PROGRAM UserMode
VAR
(*GapMode*)
	UserGapPositionNew:LREAL:=20;//target
	UserGapVelocityNew:LREAL:=0.02;//target
	UserGapPositionDisplay:LREAL;//current
	UserGapVelocityDisplay:LREAL;//current
(*ID taper mode*)
	UserTaperPositionNew:LREAL:=0;//target
	UserTaperVelocityNew:LREAL:=0.02;//target
	UserTaperPositionDisplay:LREAL;//current
	UserTaperPositionDisplayBLSide:LREAL;//current BeamLine
	UserTaperPositionActual:LREAL;//current
	UserTaperVelocityDisplay:LREAL;//target
	UserGapPositionDisplay_FromLeftTop:LREAL;
	UserGapPositionDisplay_FromLeftBottom:LREAL;
		//
	UserRightGapPositionNew:LREAL;
	UserRightGapVelocityNew:LREAL;
	UserRightGapPositionDisplay:LREAL;
	UserRightGapVelocityDisplay:LREAL;
	UserRightGapPositionDisplay_FromRightTop:LREAL;
	UserRightGapPositionDisplay_FromRightBottom:LREAL;
(*BL taper mode*)
	BLUserTaperPositionNew:LREAL:=0;//target
	BLUserTaperVelocityNew:LREAL:=0.02;//target
	BLUserTaperPositionDisplay:LREAL;//current
	//BLUserTaperPositionDisplayBLSide:LREAL;//current BeamLine
	BLUserTaperPositionActual:LREAL;//current
	BLUserTaperVelocityDisplay:LREAL;//target
	BLUserGapPositionDisplay_FromLeftTop:LREAL;
	BLUserGapPositionDisplay_FromLeftBottom:LREAL;
	//
	BLUserLeftGapPositionNew:LREAL;
	BLUserLeftGapVelocityNew:LREAL;
	BLUserLeftGapPositionDisplay:LREAL;
	BLUserLeftGapVelocityDisplay:LREAL;
	BLUserLeftGapPositionDisplay_FromLeftTop:LREAL;
	BLUserLeftGapPositionDisplay_FromLeftBottom:LREAL;
	BLUserRightGapPositionNew:LREAL;
	BLUserRightGapVelocityNew:LREAL;
	BLUserRightGapPositionDisplay:LREAL;
	BLUserRightGapVelocityDisplay:LREAL;
	BLUserRightGapPositionDisplay_FromRightTop:LREAL;
	BLUserRightGapPositionDisplay_FromRightBottom:LREAL;

	(**)
	btn_UserGapMove:BOOL;
	btn_UserGapStop:BOOL;
	(*Var*)
	fb_ton1:TON;
	fb_ton2:TON;
	fb_ton3:TON;
	(*Status*)
	State:DINT;
	Busy:BOOL;
	InitPowerDone:BOOL;
	InitCompensationDatasDone:BOOL;
	(*FB*)
	m_state: DINT;
	n_state: DINT;
	s_state: DINT;
	(*¼ì²âµ½ÏÞÎ»£¬»Ö¸´Move×´Ì¬*)
	FTrig_ReachLS: F_TRIG;
	FTrig_btn_GapMove: F_TRIG;
	GapOutRange: BOOL;
	(*PowerOff*)
	d_state: DINT;
	i: INT;
	j: INT;
	k: INT;
	moni_State:DINT;
	TargetPosLessThanCurrentPos:BOOL;
	TargetLTPosLessThanCurrentLTPos:BOOL;
	TargetRTPosLessThanCurrentRTPos:BOOL;
	TargetLBPosLessThanCurrentLBPos:BOOL;
	TargetRBPosLessThanCurrentRBPos:BOOL;
	PositiveMoving:BOOL;
	HysteresisMoving:BOOL;
	NoneHysteresisMoving:BOOL;
	(*Spectroscopy scanning Mode*)
	IsSSMotionMode:BOOL;
	RegularMotionMode:BOOL;
	SSMotionMode:BOOL;
	SS_StepSize:LREAL:=0.001;
	SS_StepNumber:INT:=10;
	SS_StepVelocity:LREAL:=1;
	SS_Move:BOOL;
	SS_Stop:BOOL;
	SS_MoveState:DINT;
	SS_StopState:DINT;
	SS_currentStep:DINT:=0;
	SS_StepSystemTime_Begin:ARRAY[0..100] OF ULINT;
	SS_StepSystemTime_End:ARRAY[0..100] OF ULINT;
	SS_StepCountTime:ARRAY[0..100] OF ULINT;
	SS_TimeCountBegin:BOOL;
	m: INT;
	SS_TON: TON;
	StepEachTime:TIME;
	StepEachTime_ms:INT:=1000;//ms
	SS_OTSTRUCT :OTSTRUCT ;
	SS_StartPositionDisplay:LREAL;
	RTRG_SS_StartPositionDisplay:R_TRIG;
	SS_InitStartPositionDone:BOOL;

	//
	min_SS_StepSize	: LREAL:=0;
	max_SS_StepSize	: LREAL:=200;
	inRange_SS_StepSize	: BOOL;
	//
	min_SS_StepNumber	: INT:=1;
	max_SS_StepNumber	: INT:=1000;
	inRange_SS_StepNumber	: BOOL;
	//
	min_SS_StepVelocity:LREAL:=0;
	max_SS_StepVelocity:LREAL:=1;
	inRange_SS_StepVelocity:BOOL;
	//
	min_StepEachTime_ms:INT:=100;
	max_StepEachTime_ms:INT:=10000;
	inRange_StepEachTime_ms:BOOL;
	l: INT;
	Threshold_UserTopPos_PLC: LREAL;
	Threshold_UserTopVelo_PLC: LREAL;
	Threshold_UserBottomPos_PLC: LREAL;
	Threshold_UserBottomVelo_PLC: LREAL;
	Threshold_UserLeftPos_PLC: LREAL;
	Threshold_UserLeftVelo_PLC: LREAL;
	Threshold_UserRightPos_PLC: LREAL;
	Threshold_UserRightVelo_PLC: LREAL;
	testa: BOOL;
	testb: BOOL;
	//Taper parameters
	Threshold_GapChangeFlag: LREAL:=0.001;
	Threshold_TaperChangeFlag: LREAL:=0.005;
	TaperAndGapSafetyfactor: LREAL:=1;
	TaperAndGapSafetyScale:LREAL:=0.41;//IAU=0.409,IVU=0.32,CPMU=0.328,IAMW=0.42
	TaperAndGapSafetyMinGapMargin:LREAL:=0.2;
	IDTaperAndBLTaperScale:LREAL:=0.548;//HU 
	//HEPSIDTaperAndBLTaperScale:LREAL:=0.55;
	//
	//Global Chain protection-MPS
	Global_ChainProtection_MPS_StorageRingReady:BOOL;
	Global_ChainProtection_MPS_On: BOOL;
	Global_ChainProtection_MPS_MaxGapValue: LREAL;
	Global_ChainProtection_MPS_MoveVelocity: LREAL;
	Global_ChainProtection_MPS_Done: BOOL;
	//Global_ChainProtection_Error: BOOL;
	//Global_ChainProtection_ErrorID: INT;
	//Global_ChainProtection_ErrorDescription: STRING;
	Global_ChainProtection_MPS_ManualOperation:BOOL:=TRUE;
	Global_ChainProtection_MPS_FTRIG:F_TRIG;
	Global_ChainProtection_MPS_FTRIG_Manul:F_TRIG;
	Global_ChainProtection_MPS_TON:TON;
	Global_ChainProtection_MPS_Triggered:BOOL;
	Global_ChainProtection_MPS_In:BOOL;
	Global_ChainProtection_MPS_In1 AT%I* :BOOL;//下降沿表示触发,EL1008
	Global_ChainProtection_MPS_In2 AT%I* :BOOL;
	Global_ChainProtection_MPS_State:DINT;
	Global_ChainProtection_MPS_Out1 AT%Q* :BOOL;//上升沿标识到达最大间隙，连锁保护成功,EL2624
	Global_ChainProtection_MPS_Out2 AT%Q* :BOOL;
	Global_ChainProtection_MPS_TON_Stop2Move:TON;
	Global_ChainProtection_MPS_TON_Stop2Move_InTaperMode:TON;
	Global_ChainProtection_MPS_TON_Power2Move:TON;
	//Global Chain protection-EPS
	Global_ChainProtection_EPS_BeamLineReady:BOOL;
	Global_ChainProtection_EPS_On: BOOL;
	Global_ChainProtection_EPS_MaxGapValue: LREAL;
	Global_ChainProtection_EPS_MoveVelocity: LREAL;
	Global_ChainProtection_EPS_Done: BOOL;
	//Global_ChainProtection_Error: BOOL;
	//Global_ChainProtection_ErrorID: INT;
	//Global_ChainProtection_ErrorDescription: STRING;
	Global_ChainProtection_EPS_ManualOperation:BOOL:=TRUE;
	Global_ChainProtection_EPS_FTRIG:F_TRIG;
	Global_ChainProtection_EPS_FTRIG_Manul:F_TRIG;
	Global_ChainProtection_EPS_TON:TON;
	Global_ChainProtection_EPS_Triggered:BOOL;
	Global_ChainProtection_EPS_In:BOOL;
	Global_ChainProtection_EPS_In1 AT%I* :BOOL;//下降沿表示触发,EL1124
	Global_ChainProtection_EPS_In2 AT%I* :BOOL;
	Global_ChainProtection_EPS_State:DINT;
	Global_ChainProtection_EPS_Out1 AT%Q* :BOOL;//上升沿标识到达最大间隙，连锁保护成功,EL2124
	Global_ChainProtection_EPS_Out2 AT%Q* :BOOL;
	Global_ChainProtection_EPS_TON_Stop2Move:TON;
	Global_ChainProtection_EPS_TON_Stop2Move_InTaperMode:TON;
	Global_ChainProtection_EPS_TON_Power2Move:TON;
	//
	//Cryogenic Chain protection
	Cryogenic_ChainProtection_On: BOOL;
	Cryogenic_ChainProtection_MaxGapValue: LREAL;
	Cryogenic_ChainProtection_MoveVelocity: LREAL;
	Cryogenic_ChainProtection_Done: BOOL;
	//Cryogenic_ChainProtection_Error: BOOL;
	//Cryogenic_ChainProtection_ErrorID: INT;
	//Cryogenic_ChainProtection_ErrorDescription: STRING;
	Cryogenic_ChainProtection_ManualOperation:BOOL:=TRUE;
	Cryogenic_ChainProtection_FTRIG:F_TRIG;
	Cryogenic_ChainProtection_FTRIG_Manul:F_TRIG;
	Cryogenic_ChainProtection_TON:TON;
	Cryogenic_ChainProtection_Triggered:BOOL;
	Cryogenic_ChainProtection_In:BOOL;
	Cryogenic_ChainProtection_State:DINT;
	Cryogenic_ChainProtection_Out1 AT%Q* :BOOL;//上升沿标识到达最大间隙，连锁保护成功
	Cryogenic_ChainProtection_TON_Stop2Move:TON;
	Cryogenic_ChainProtection_TON_Stop2Move_InTaperMode:TON;
	Cryogenic_ChainProtection_TON_Power2Move:TON;
	test11:INT:=1;
	IsTest11OrNot:BOOL;
	tesetBegin: BOOL;
	Threshold_motorsTargetPosCalculate: LREAL;
	SS_Stop2: BOOL;
	//
	LeftTopLinPositionNewTemp: LREAL;
	RightTopLinPositionNewTemp: LREAL;
	LeftBottomLinPositionNewTemp: LREAL;
	RightBottomLinPositionNewTemp: LREAL;
	
	
	//OneKeyToMaxGap
	btn_OneKeyToMaxGap:BOOL;
	OneKeyToMaxGap_RTRIG:R_TRIG;
	OneKeyToMaxGap_TON:TON;
	OneKeyToMaxGap_Triggered:BOOL;
	OneKeyToMaxGap_State:DINT;
	OneKeyToMaxGap_TON_Stop2Move:TON;
	OneKeyToMaxGap_TON_Stop2Move_InTaperMode:TON;
	OneKeyToMaxGap_TON_Power2Move:TON;
	OneKeyToMaxGap_Done:BOOL;
	FTrig_ReachLSa: F_TRIG;
	Unreach_LS_Fara: BOOL;
	Unreach_LS_Neara: BOOL;
	btn_UserGapStopa: BOOL;
	
	//OneKeyToMTaperZero
	btn_OneKeyToTaperZero:BOOL;
	OneKeyToTaperZero_RTRIG:R_TRIG;
	OneKeyToTaperZero_TON:TON;
	OneKeyToTaperZero_Triggered:BOOL;
	OneKeyToTaperZero_State:DINT;
	OneKeyToTaperZero_Done:BOOL;
	OneKeyToTaperZero_Delay:TON;
	//BLTaper
	CurrentTaperInit: LREAL;
	L_HalfGirder:LREAL:=2500;
	L_Center2Motor:LREAL:=1375;
	
	trig_TaperOrNot: R_TRIG;
	trig_BLTaperOrNot: R_TRIG;
END_VAR

IF NOT PositionBiasDone THEN
	RETURN;
END_IF
IF NOT loadParametersDone THEN
	RETURN;
END_IF
(*btn_Power On/Off*)
IF btn_Power AND NOT st_Power THEN
	btn_PowerOn:=TRUE;
	btn_Power:=FALSE;
END_IF
IF btn_Power AND st_Power THEN
	btn_PowerOff:=TRUE;
	btn_Power:=FALSE;
END_IF
IF btn_PowerOn THEN
	A_PowerOn();
END_IF
IF btn_PowerOff THEN
	A_PowerOff();
END_IF

(*检查couple状态，不允许couple*)
A_CheckCoupleStatus();

(*监控四轴位置速度等*)
A_MonitoringAllAxis();

(*目标位置和速度保护*)
A_CheckMotorsPos();

(*补偿数据处理*)
A_InitCompensationData();

(*常规磁间隙开合*)
IF RegularMotionMode AND NOT SSMotionMode THEN
	A_RegularMotion();
END_IF

(*Spectroscopy scanning Mode*)
IF IsSSMotionMode THEN
	SSMotionMode:=TRUE;
	RegularMotionMode:=FALSE;
ELSE
	SSMotionMode:=FALSE;
	RegularMotionMode:=TRUE;
END_IF
IF	SSMotionMode AND NOT RegularMotionMode THEN
	A_SpectroscopyScanningMotion();
END_IF


(*GlobalChainProtection*)
A_GlobalChainProtection_MPS();
A_GlobalChainProtection_EPS();

(*CryogenicChainProtection*)
A_CryogenicChainProtection();

(*A_OneKeyToMaxGap*)
A_OneKeyToMaxGap();

(*A_OneKeyToTaperZero*)
A_OneKeyToTaperZero();

(*A_TaperParametersInit*)
A_TaperParametersInit();

ACTION A_CheckCoupleStatus:
IF NOT btn_PowerOff THEN
	IF st_Power=1 AND st_Couple<>0THEN
		Error:=TRUE;
		ErrorID:=501;
		LeftTopLinMoveIndicator:=0;
		RightTopLinMoveIndicator:=0;
		LeftBottomLinMoveIndicator:=0;
		RightBottomLinMoveIndicator:=0;
		FB_PlcEmergencyStop();
		LED_Error:=TRUE;
		ErrorDescription:='couple stutas error';
	END_IF
END_IF
END_ACTION

ACTION A_CheckMotorsPos:
//
//目标位置速度超出阈值判断
//
//gap posiion
IF UserGapPositionNew<min_UserGapPositionNew OR UserGapPositionNew>max_UserGapPositionNew THEN
	inRange_UserGapPositionNew:=FALSE;
END_IF
IF UserGapPositionNew>=min_UserGapPositionNew AND UserGapPositionNew<=max_UserGapPositionNew THEN
	inRange_UserGapPositionNew:=TRUE;
END_IF
//gap velocity
IF UserGapVelocityNew<min_UserGapVelocityNew OR UserGapVelocityNew>max_UserGapVelocityNew THEN
	inRange_UserGapVelocityNew:=FALSE;
END_IF
IF UserGapVelocityNew>=min_UserGapVelocityNew AND UserGapVelocityNew<=max_UserGapVelocityNew THEN
	inRange_UserGapVelocityNew:=TRUE;
END_IF
//taper position
IF UserTaperPositionNew<min_UserTaperPositionNew OR UserTaperPositionNew>max_UserTaperPositionNew THEN
	inRange_UserTaperPositionNew:=FALSE;
END_IF
IF UserTaperPositionNew>=min_UserTaperPositionNew AND UserTaperPositionNew<=max_UserTaperPositionNew THEN
	inRange_UserTaperPositionNew:=TRUE;
END_IF
//taper velocity
IF UserTaperVelocityNew<min_UserTaperVelocityNew OR UserTaperVelocityNew>max_UserTaperVelocityNew THEN
	inRange_UserTaperVelocityNew:=FALSE;
END_IF
IF UserTaperVelocityNew>=min_UserTaperVelocityNew AND UserTaperVelocityNew<=max_UserTaperVelocityNew THEN
	inRange_UserTaperVelocityNew:=TRUE;
END_IF
//SS Mode
IF SS_StepSize<min_SS_StepSize OR SS_StepSize>max_SS_StepSize THEN
	inRange_SS_StepSize:=FALSE;
END_IF
IF SS_StepSize>=min_SS_StepSize AND SS_StepSize<=max_SS_StepSize THEN
	inRange_SS_StepSize:=TRUE;
END_IF
IF SS_StepNumber<min_SS_StepNumber OR SS_StepNumber>max_SS_StepNumber THEN
	inRange_SS_StepNumber:=FALSE;
END_IF
IF SS_StepNumber>=min_SS_StepNumber AND SS_StepNumber<=max_SS_StepNumber THEN
	inRange_SS_StepNumber:=TRUE;
END_IF
IF SS_StepVelocity<min_SS_StepVelocity OR SS_StepVelocity>max_SS_StepVelocity THEN
	inRange_SS_StepVelocity:=FALSE;
END_IF
IF SS_StepVelocity>=min_SS_StepVelocity AND SS_StepVelocity<=max_SS_StepVelocity THEN
	inRange_SS_StepVelocity:=TRUE;
END_IF
IF StepEachTime_ms<min_StepEachTime_ms OR StepEachTime_ms>max_StepEachTime_ms THEN
	inRange_StepEachTime_ms:=FALSE;
END_IF
IF StepEachTime_ms>=min_StepEachTime_ms AND StepEachTime_ms<=max_StepEachTime_ms THEN
	inRange_StepEachTime_ms:=TRUE;
END_IF


//
//输入速度和位置保护
//
IF btn_UserGapMove  AND NOT SSMotionMode AND RegularMotionMode THEN
	IF NOT inRange_UserGapPositionNew THEN
		btn_UserGapStop:=TRUE;
		btn_UserGapMove:=FALSE;
		Error:=TRUE;
		ErrorId:=801;
		ErrorDescription:='target Gap position out of range,please check';
		RETURN;
	ELSE
		//btn_UserGapStop:=FALSE;
		Error:=FALSE;
		ErrorId:=0;
		ErrorDescription:='';	
	END_IF
	IF NOT inRange_UserGapVelocityNew THEN
		btn_UserGapStop:=TRUE;
		btn_UserGapMove:=FALSE;
		Error:=TRUE;
		ErrorId:=802;
		ErrorDescription:='target Gap velocity out of range,please check';
		RETURN;
	ELSE
		//btn_UserGapStop:=FALSE;
		Error:=FALSE;
		ErrorId:=0;
		ErrorDescription:='';
	END_IF
	IF NOT inRange_UserTaperPositionNew THEN
		btn_UserGapStop:=TRUE;
		btn_UserGapMove:=FALSE;
		Error:=TRUE;
		ErrorId:=803;
		ErrorDescription:='target Taper Position out of range,please check';
		RETURN;
	ELSE
		//btn_UserGapStop:=FALSE;
		Error:=FALSE;
		ErrorId:=0;
		ErrorDescription:='';
	END_IF
	IF NOT inRange_UserTaperVelocityNew THEN
		btn_UserGapStop:=TRUE;
		btn_UserGapMove:=FALSE;
		Error:=TRUE;
		ErrorId:=804;
		ErrorDescription:='target Taper velocity out of range,please check';
		RETURN;
	ELSE
		//btn_UserGapStop:=FALSE;
		Error:=FALSE;
		ErrorId:=0;
		ErrorDescription:='';
	END_IF
END_IF

//
//运动过程中，监控目标位置速度
//
IF moveStatusAnyAxis THEN
	IF NOT inRange_UserGapPositionNew THEN
		btn_UserGapStop:=TRUE;
		Error:=TRUE;
		ErrorId:=805;
		ErrorDescription:='target Gap position out of range in moving process!';
		FB_PlcEmergencyStop();
	END_IF
	IF NOT inRange_UserGapVelocityNew THEN
		btn_UserGapStop:=TRUE;
		Error:=TRUE;
		ErrorId:=806;
		ErrorDescription:='target Gap velocity out of range in moving process!';
		FB_PlcEmergencyStop();
	END_IF
	IF NOT inRange_UserTaperPositionNew THEN
		btn_UserGapStop:=TRUE;
		Error:=TRUE;
		ErrorId:=807;
		ErrorDescription:='target Taper Position out of range in moving process!';
		FB_PlcEmergencyStop();
	END_IF
	IF NOT inRange_UserTaperVelocityNew THEN
		btn_UserGapStop:=TRUE;
		Error:=TRUE;
		ErrorId:=808;
		ErrorDescription:='target Taper velocity out of range in moving process!';
		FB_PlcEmergencyStop();
	END_IF
END_IF
//
//运动过程中，监控每一个轴的目标位置，目标位置若超出阈值，Emergency
//
IF moveStatusAnyAxis THEN
	IF NOT TaperOrNot THEN
		IF LeftTopLinPositionNew<min_UserLEProtectionGapPosition/2 OR LeftTopLinPositionNew>max_UserLEProtectionGapPosition/2 THEN
			btn_UserGapStop:=TRUE;
			Error:=TRUE;
			ErrorId:=809;
			ErrorDescription:='target LeftTop position out of range in moving process!';
			FB_PlcEmergencyStop();
		END_IF
		IF RightTopLinPositionNew<min_UserLEProtectionGapPosition/2 OR RightTopLinPositionNew>max_UserLEProtectionGapPosition/2 THEN
			btn_UserGapStop:=TRUE;
			Error:=TRUE;
			ErrorId:=810;
			ErrorDescription:='target RightTop velocity out of range in moving process!';
			FB_PlcEmergencyStop();
		END_IF
		IF LeftBottomLinPositionNew<min_UserLEProtectionGapPosition/2 OR LeftBottomLinPositionNew>max_UserLEProtectionGapPosition/2 THEN
			btn_UserGapStop:=TRUE;
			Error:=TRUE;
			ErrorId:=812;
			ErrorDescription:='target LeftBottom Position out of range in moving process!';
			FB_PlcEmergencyStop();
		END_IF
		IF RightBottomLinPositionNew<min_UserLEProtectionGapPosition/2 OR RightBottomLinPositionNew>max_UserLEProtectionGapPosition/2 THEN
			btn_UserGapStop:=TRUE;
			Error:=TRUE;
			ErrorId:=813;
			ErrorDescription:='target RightBottom Position out of range in moving process!';
			FB_PlcEmergencyStop();
		END_IF
	ELSE//Taper状态的保护
		;//Taper状态下，不用监控四轴位置，只需要监控目标Taper位置。在上面已经保护
	END_IF
END_IF
END_ACTION

ACTION A_CryogenicChainProtection:
//总开关
IF NOT Cryogenic_ChainProtection_On THEN
	RETURN;
END_IF
IF NOT MAIN.CryogenicCompensationOn THEN
	RETURN;
END_IF
//判断插入件状态，是否就位
//IF NOT IDControlReady THEN
//	Cryogenic_ChainProtection_Done:=FALSE;
//	Error:= TRUE;
//	ErrorID:=1501;
//	ErrorDescription:='ID NOT READY!';
//	RETURN;
//END_IF

//
//全局连锁保护程序开始
//
//0.检测温度变化超出正常范围，或者手动触发，触发低温联锁保护
//1.判断电机是否在开启状态,没有就打开电源
//2.判断是否在Moving状态,若有就Stop
//3.将磁间隙打开到至最大阈值
//4.到位后给出反馈，且安全PLC触发
//IF MAIN.temperatureStatus=3 THEN //=2低温,超出低温阈值就触发保护
//	Cryogenic_ChainProtection_Triggered:=TRUE;
//END_IF
Cryogenic_ChainProtection_FTRIG(CLK:=MAIN.InCryogenicOrNot);
IF Cryogenic_ChainProtection_FTRIG.Q THEN
	Cryogenic_ChainProtection_Triggered:=TRUE;
END_IF
Cryogenic_ChainProtection_FTRIG_Manul(CLK:=Cryogenic_ChainProtection_ManualOperation);
IF Cryogenic_ChainProtection_FTRIG_Manul.Q THEN
	Cryogenic_ChainProtection_Triggered:=TRUE;
END_IF
IF Cryogenic_ChainProtection_Triggered THEN
	//判断当前间隙，如果比Cryogenic_ChainProtection_MaxGapValue大，则不动作，只报警，且安全PLC触发
	IF UserGapPositionDisplay - Cryogenic_ChainProtection_MaxGapValue >=0.001THEN
		Cryogenic_ChainProtection_Done:=TRUE;
		Plc_EmergencyStop:=FALSE;
		Error:= TRUE;
		ErrorID:= 1502;
		ErrorDescription:='Cryogenic Abnormal !';
		RETURN;
	END_IF
	CASE Cryogenic_ChainProtection_State OF
		0://1.判断电机是否在开启状态,没有就打开电源
			IF st_Power=1 THEN
				Cryogenic_ChainProtection_State:=1;
			ELSE
				btn_PowerOn:=TRUE;
				IF btn_PowerOn THEN
					A_PowerOn();
				END_IF
			END_IF
		1://1.判断是否在谱学扫描模式，如果是，则切换回正常运动模式
			IF IsSSMotionMode THEN
				SS_Stop:=TRUE;
				IsSSMotionMode:=FALSE;
			END_IF
			Cryogenic_ChainProtection_State:=2;
		2://判断是否在taper，如果在taper,则判断是否在运动，如果是，则停止运动,0.5sh后，转入下一步
			IF TaperOrNot THEN
				IF moveStatusLeftTop OR moveStatusRightTop OR moveStatusLeftBottom OR moveStatusRightBottom THEN
					btn_UserGapStop:=TRUE;
				ELSE
					Cryogenic_ChainProtection_TON_Stop2Move_InTaperMode(PT:=T#0.5S);
					Cryogenic_ChainProtection_TON_Stop2Move_InTaperMode.IN:=TRUE;
					IF Cryogenic_ChainProtection_TON_Stop2Move_InTaperMode.Q THEN
						TaperOrNot:=FALSE;//关闭taper模式
						Cryogenic_ChainProtection_State:=3;
					END_IF
				END_IF
			ELSE
				Cryogenic_ChainProtection_State:=3;
			END_IF
		3://3.判断是否在Moving状态,若有就Stop.Taper模式已处理完，此处开始走正常GAP开合逻辑
			IF moveStatusLeftTop OR moveStatusRightTop OR moveStatusLeftBottom OR moveStatusRightBottom THEN
				btn_UserGapStop:=TRUE;
			ELSE
				Cryogenic_ChainProtection_TON_Stop2Move(PT:=T#0.5S);
				Cryogenic_ChainProtection_TON_Stop2Move.IN:=TRUE;
				IF Cryogenic_ChainProtection_TON_Stop2Move.Q THEN
					Cryogenic_ChainProtection_State:=4;
				END_IF
			END_IF
		4://4.将磁间隙打开到至最大阈值
			Cryogenic_ChainProtection_TON(PT:=INT_TO_TIME(LREAL_TO_INT(Cryogenic_ChainProtection_MaxGapValue/Cryogenic_ChainProtection_MoveVelocity+30))*1000);
			Cryogenic_ChainProtection_TON.IN:=TRUE;
			Cryogenic_ChainProtection_TON_Power2Move(PT:=T#0.1S);
			Cryogenic_ChainProtection_TON_Power2Move.IN:=TRUE;
			UserGapPositionNew:=Cryogenic_ChainProtection_MaxGapValue;
			UserGapVelocityNew:=Cryogenic_ChainProtection_MoveVelocity;
			btn_UserGapMove:=TRUE;
			IF Cryogenic_ChainProtection_TON_Power2Move.Q THEN
				IF FB_MOVE.BCGapDone THEN
					Cryogenic_ChainProtection_State:=88;
				END_IF
			END_IF
			IF Cryogenic_ChainProtection_TON.Q THEN//如果150s后，还没有运动到指定gap，则报错
				Cryogenic_ChainProtection_State:=-100;
			END_IF
		88://4.到位后给出反馈，且安全PLC触发
			Cryogenic_ChainProtection_Done:=TRUE;
			Plc_EmergencyStop:=FALSE;		
			Error:=TRUE;
			ErrorID:=1503;
			ErrorDescription:='Cryogenic_ChainProtection Triggered';
		-100:
			Cryogenic_ChainProtection_Done:=FALSE;
			Error:=TRUE;
			ErrorID:=1504;
			ErrorDescription:='NOT MOVING TO MAXGAP';
	END_CASE
END_IF

//监控是否同时是低温模式，且温度传感器检测到的是低温+10℃（避开低温联锁保护，联锁保护要求在低温阈值时拉开磁间隙）
IF MAIN.temperatureStatus<>0 AND MAIN.temperature_average > MAIN.CryogenicTemperatureThreshold +10 THEN//在低温+10℃
	IF MAIN.HasTemperatureSensorOrNot AND MAIN.CryogenicCompensationOn THEN
			Error:=TRUE;
			ErrorID:=1505;
			Plc_EmergencyStop:=FALSE;
			ErrorDescription:='CryogenicCompensationOn AND Room temperatureStatus';
	END_IF
END_IF
END_ACTION

ACTION A_GlobalChainProtection_EPS:
//硬线输入定义
Global_ChainProtection_EPS_In:=Global_ChainProtection_EPS_In1 AND Global_ChainProtection_EPS_In2;
//硬线输出定义
Global_ChainProtection_EPS_Out1:=Global_ChainProtection_EPS_Done;
Global_ChainProtection_EPS_Out2:=Global_ChainProtection_EPS_Done;
//总开关
IF NOT Global_ChainProtection_EPS_On THEN
	RETURN;
END_IF
//判断插入件状态，是否就位
//IF NOT IDControlReady THEN
//	Global_ChainProtection_EPS_Done:=FALSE;
//	Error:= TRUE;
//	ErrorID:= 1501;
//	ErrorDescription:='ID NOT READY!';
//	RETURN;
//END_IF
//判断储存环是否给出就位信号，暂时由参数表给出TRUE，最终将由IOC接受PV
IF 	NOT Global_ChainProtection_EPS_BeamLineReady THEN
	Global_ChainProtection_EPS_Done:=FALSE;
	Error:= TRUE;
	ErrorID:= 1503;
	ErrorDescription:='Global_ChainProtection_EPS_BeamLineReady NOT Ready';
	RETURN;
END_IF
//
//全局连锁保护程序开始
//
//0.检测到下降沿，触发
//1.判断电机是否在开启状态,没有就打开电源
//2.判断是否在Moving状态,若有就Stop
//3.将磁间隙打开到至最大阈值
//4.到位后给出反馈，且安全PLC触发
Global_ChainProtection_EPS_FTRIG(CLK:=Global_ChainProtection_EPS_In);
IF Global_ChainProtection_EPS_FTRIG.Q THEN
	Global_ChainProtection_EPS_Triggered:=TRUE;
END_IF
Global_ChainProtection_EPS_FTRIG_Manul(CLK:=Global_ChainProtection_EPS_ManualOperation);
IF Global_ChainProtection_EPS_FTRIG_Manul.Q THEN
	Global_ChainProtection_EPS_Triggered:=TRUE;
END_IF
IF Global_ChainProtection_EPS_Triggered THEN
	CASE Global_ChainProtection_EPS_State OF
		0://1.判断电机是否在开启状态,没有就打开电源
			IF st_Power=1 THEN
				Global_ChainProtection_EPS_State:=1;
			ELSE
				btn_PowerOn:=TRUE;
				IF btn_PowerOn THEN
					A_PowerOn();
				END_IF
			END_IF
		1://1.判断是否在谱学扫描模式，如果是，则切换回正常运动模式
			IF IsSSMotionMode THEN
				SS_Stop:=TRUE;
				IsSSMotionMode:=FALSE;
			END_IF
			Global_ChainProtection_EPS_State:=2;
		2://判断是否在taper，如果在taper,则判断是否在运动，如果是，则停止运动,0.5sh后，转入下一步
			IF TaperOrNot THEN
				IF moveStatusLeftTop OR moveStatusRightTop OR moveStatusLeftBottom OR moveStatusRightBottom THEN
					btn_UserGapStop:=TRUE;
				ELSE
					Global_ChainProtection_EPS_TON_Stop2Move_InTaperMode(PT:=T#0.5S);
					Global_ChainProtection_EPS_TON_Stop2Move_InTaperMode.IN:=TRUE;
					IF Global_ChainProtection_EPS_TON_Stop2Move_InTaperMode.Q THEN
						TaperOrNot:=FALSE;//关闭taper模式
						Global_ChainProtection_EPS_State:=3;
					END_IF
				END_IF
			ELSE
				Global_ChainProtection_EPS_State:=3;
			END_IF
		3://3.判断是否在Moving状态,若有就Stop.Taper模式已处理完，此处开始走正常GAP开合逻辑
			IF moveStatusLeftTop OR moveStatusRightTop OR moveStatusLeftBottom OR moveStatusRightBottom THEN
				btn_UserGapStop:=TRUE;
			ELSE
				Global_ChainProtection_EPS_TON_Stop2Move(PT:=T#0.5S);
				Global_ChainProtection_EPS_TON_Stop2Move.IN:=TRUE;
				IF Global_ChainProtection_EPS_TON_Stop2Move.Q THEN
					Global_ChainProtection_EPS_State:=4;
				END_IF
			END_IF
		4://当前磁间隙如何和最大磁间隙差别不大，不超过0.1，则直接保护
			IF ABS(UserGapPositionDisplay-Global_ChainProtection_EPS_MaxGapValue)<=0.1 THEN
				Global_ChainProtection_EPS_Done:=TRUE;
				Plc_EmergencyStop:=FALSE;	
				Error:=TRUE;
				ErrorID:=1506;
				ErrorDescription:='EPS Triggered,but ABS(GapPositionDisplay-EPS_MaxGapValue)<=0.1 ';	
			ELSE
				Global_ChainProtection_EPS_State:=5;
			END_IF
		5://5.将磁间隙打开到至最大阈值
			Global_ChainProtection_EPS_TON(PT:=INT_TO_TIME(LREAL_TO_INT(Global_ChainProtection_EPS_MaxGapValue/Global_ChainProtection_EPS_MoveVelocity+30))*1000);
			Global_ChainProtection_EPS_TON.IN:=TRUE;
			Global_ChainProtection_EPS_TON_Power2Move(PT:=T#0.1S);
			Global_ChainProtection_EPS_TON_Power2Move.IN:=TRUE;
			UserGapPositionNew:=Global_ChainProtection_EPS_MaxGapValue;
			UserGapVelocityNew:=Global_ChainProtection_EPS_MoveVelocity;
			btn_UserGapMove:=TRUE;
			IF Global_ChainProtection_EPS_TON_Power2Move.Q THEN
				IF FB_MOVE.BCGapDone THEN
					Global_ChainProtection_EPS_State:=88;
				END_IF
			END_IF
			IF Global_ChainProtection_EPS_TON.Q THEN//如果150s后，还没有运动到指定gap，则报错
				Global_ChainProtection_EPS_State:=-100;
			END_IF
		88://6.到位后给出反馈，且安全PLC触发
			Global_ChainProtection_EPS_Done:=TRUE;
			Plc_EmergencyStop:=FALSE;	
			Error:=TRUE;
			ErrorID:=1504;
			ErrorDescription:='Global_ChainProtection_EPS Triggered ';	
		-100:
			Global_ChainProtection_EPS_Done:=FALSE;
			Error:=TRUE;
			ErrorID:=1505;
			ErrorDescription:='NOT MOVING TO MAXGAP';
	END_CASE
END_IF
END_ACTION

ACTION A_GlobalChainProtection_MPS:
//硬线输入定义
Global_ChainProtection_MPS_In:=Global_ChainProtection_MPS_In1 AND Global_ChainProtection_MPS_In2;
//硬线输出定义
Global_ChainProtection_MPS_Out1:=Global_ChainProtection_MPS_Done;
Global_ChainProtection_MPS_Out2:=Global_ChainProtection_MPS_Done;
//总开关
IF NOT Global_ChainProtection_MPS_On THEN
	RETURN;
END_IF
//判断插入件状态，是否就位
//IF NOT IDControlReady THEN
//	Global_ChainProtection_MPS_Done:=FALSE;
//	Error:= TRUE;
//	ErrorID:= 1401;
//	ErrorDescription:='ID NOT READY!';
//	RETURN;
//END_IF
//判断储存环是否给出就位信号，暂时由参数表给出TRUE，最终将由IOC接受PV
IF 	NOT Global_ChainProtection_MPS_StorageRingReady THEN
	Global_ChainProtection_MPS_Done:=FALSE;
	Error:= TRUE;
	ErrorID:= 1403;
	ErrorDescription:='StorageRingChainProtection NOT Ready';
	RETURN;
END_IF
//
//全局连锁保护程序开始
//
//0.检测到下降沿，触发
//1.判断电机是否在开启状态,没有就打开电源
//2.判断是否在Moving状态,若有就Stop
//3.将磁间隙打开到至最大阈值
//4.到位后给出反馈，且安全PLC触发
Global_ChainProtection_MPS_FTRIG(CLK:=Global_ChainProtection_MPS_In);
IF Global_ChainProtection_MPS_FTRIG.Q THEN
	Global_ChainProtection_MPS_Triggered:=TRUE;
END_IF
Global_ChainProtection_MPS_FTRIG_Manul(CLK:=Global_ChainProtection_MPS_ManualOperation);
IF Global_ChainProtection_MPS_FTRIG_Manul.Q THEN
	Global_ChainProtection_MPS_Triggered:=TRUE;
END_IF
IF Global_ChainProtection_MPS_Triggered THEN
	CASE Global_ChainProtection_MPS_State OF
		0://1.判断电机是否在开启状态,没有就打开电源
			IF st_Power=1 THEN
				Global_ChainProtection_MPS_State:=1;
			ELSE
				btn_PowerOn:=TRUE;
				IF btn_PowerOn THEN
					A_PowerOn();
				END_IF
			END_IF
		1://1.判断是否在谱学扫描模式，如果是，则切换回正常运动模式
			IF IsSSMotionMode THEN
				SS_Stop:=TRUE;
				IsSSMotionMode:=FALSE;
			END_IF
			Global_ChainProtection_MPS_State:=2;
		2://判断是否在taper，如果在taper,则判断是否在运动，如果是，则停止运动,0.5sh后，转入下一步
			IF TaperOrNot THEN
				IF moveStatusLeftTop OR moveStatusRightTop OR moveStatusLeftBottom OR moveStatusRightBottom THEN
					btn_UserGapStop:=TRUE;
				ELSE
					Global_ChainProtection_MPS_TON_Stop2Move_InTaperMode(PT:=T#0.5S);
					Global_ChainProtection_MPS_TON_Stop2Move_InTaperMode.IN:=TRUE;
					IF Global_ChainProtection_MPS_TON_Stop2Move_InTaperMode.Q THEN
						TaperOrNot:=FALSE;//关闭taper模式
						Global_ChainProtection_MPS_State:=3;
					END_IF
				END_IF
			ELSE
				Global_ChainProtection_MPS_State:=3;
			END_IF
		3://3.判断是否在Moving状态,若有就Stop.Taper模式已处理完，此处开始走正常GAP开合逻辑
			IF moveStatusLeftTop OR moveStatusRightTop OR moveStatusLeftBottom OR moveStatusRightBottom THEN
				btn_UserGapStop:=TRUE;
			ELSE
				Global_ChainProtection_MPS_TON_Stop2Move(PT:=T#0.5S);
				Global_ChainProtection_MPS_TON_Stop2Move.IN:=TRUE;
				IF Global_ChainProtection_MPS_TON_Stop2Move.Q THEN
					Global_ChainProtection_MPS_State:=4;
				END_IF
			END_IF
		4://当前磁间隙如何和最大磁间隙差别不大，不超过0.1，则直接保护
			IF ABS(UserGapPositionDisplay-Global_ChainProtection_MPS_MaxGapValue)<=0.1 THEN
				Global_ChainProtection_MPS_Done:=TRUE;
				Plc_EmergencyStop:=FALSE;	
				Error:=TRUE;
				ErrorID:=1406;
				ErrorDescription:='MPS Triggered,but ABS(GapPositionDisplay-MPS_MaxGapValue)<=0.1 ';	
			ELSE
				Global_ChainProtection_MPS_State:=5;
			END_IF
		5://5.将磁间隙打开到至最大阈值
			Global_ChainProtection_MPS_TON(PT:=INT_TO_TIME(LREAL_TO_INT(Global_ChainProtection_MPS_MaxGapValue/Global_ChainProtection_MPS_MoveVelocity+30))*1000);
			Global_ChainProtection_MPS_TON.IN:=TRUE;
			Global_ChainProtection_MPS_TON_Power2Move(PT:=T#0.1S);
			Global_ChainProtection_MPS_TON_Power2Move.IN:=TRUE;
			UserGapPositionNew:=Global_ChainProtection_MPS_MaxGapValue;
			UserGapVelocityNew:=Global_ChainProtection_MPS_MoveVelocity;
			btn_UserGapMove:=TRUE;
			IF Global_ChainProtection_MPS_TON_Power2Move.Q THEN
				IF FB_MOVE.BCGapDone THEN
					Global_ChainProtection_MPS_State:=88;
				END_IF
			END_IF
			IF Global_ChainProtection_MPS_TON.Q THEN//如果150s后，还没有运动到指定gap，则报错
				Global_ChainProtection_MPS_State:=-100;
			END_IF
		88://6.到位后给出反馈，且安全PLC触发
			Global_ChainProtection_MPS_Done:=TRUE;
			Plc_EmergencyStop:=FALSE;	
			Error:=TRUE;
			ErrorID:=1404;
			ErrorDescription:='Global_ChainProtection_MPS Triggered ';	
		-100:
			Global_ChainProtection_MPS_Done:=FALSE;
			Error:=TRUE;
			ErrorID:=1405;
			ErrorDescription:='NOT MOVING TO MAXGAP';
	END_CASE
END_IF
END_ACTION

ACTION A_InitCompensationData:
(*补偿开始*)
IF USE_SingleAxis_Compensation THEN
(*正常gap模式以及插入件taper模式下，只运动出口电机，因此只解算出口位置*)
	IF NormalGapMode OR IDTaperMode THEN
		//
		//1.目标位置解算
		//
		(*通过补偿表解算四轴目标位置*)
		//左轴位置由Gap定，右轴位置由右gap定。右gap值=左gap+taper。taper模式和非taper模式一样，非taper模式只是一种特例存在
		//左轴目标位置解算
		IF NOT TaperOrNot THEN
			UserTaperPositionNew:=0;
			//UserTaperPositionDisplay:=0;
		END_IF
		UserRightGapPositionNew:=UserGapPositionNew+UserTaperPositionNew;
		//左轴目标位置解算
		FOR	i:= 1 TO 17 DO
				IF UserGapPositionNew/2<M_Compensation[i+1].Encoder AND UserGapPositionNew/2>=M_Compensation[i].Encoder THEN
					IF i<>18 THEN
						LeftTopLinPositionNew:=(((UserGapPositionNew/2-M_Compensation[i].Encoder)*(M_Compensation[i+1].LeftTop-M_Compensation[i].LeftTop))
								/(M_Compensation[i+1].Encoder-M_Compensation[i].Encoder))+M_Compensation[i].LeftTop;
						LeftBottomLinPositionNew:=(((UserGapPositionNew/2-M_Compensation[i].Encoder)*(M_Compensation[i+1].LeftBottom-M_Compensation[i].LeftBottom))
								/(M_Compensation[i+1].Encoder-M_Compensation[i].Encoder))+M_Compensation[i].LeftBottom;
						M_CompensationNumber:=i;
						InitCompensationDatasDone:=TRUE;
					ELSIF i=18 AND UserGapPositionNew/2=M_Compensation[i].Encoder THEN		(*Gap=14µÄÌØÊâÇé¿ö*)
						(**)
						LeftTopLinPositionNew:=M_Compensation[i].LeftTop;
						LeftBottomLinPositionNew:=M_Compensation[i].LeftBottom;
						M_CompensationNumber:=i;
						InitCompensationDatasDone:=TRUE;
					ELSE
						LeftTopLinPositionNew:=UserGapPositionNew/2;
						LeftBottomLinPositionNew:=UserGapPositionNew/2;
						M_CompensationNumber:=i;
						InitCompensationDatasDone:=TRUE;
					END_IF
				END_IF
		END_FOR
		//右轴目标位置解算
		FOR	j:= 1 TO 17 DO
			IF UserRightGapPositionNew/2<M_Compensation[j+1].Encoder AND UserRightGapPositionNew/2>=M_Compensation[j].Encoder THEN
				IF j<>18 THEN
					RightTopLinPositionNew:=(((UserRightGapPositionNew/2-M_Compensation[j].Encoder)*(M_Compensation[j+1].RightTop-M_Compensation[j].RightTop))
							/(M_Compensation[j+1].Encoder-M_Compensation[j].Encoder))+M_Compensation[j].RightTop;
					RightBottomLinPositionNew:=(((UserRightGapPositionNew/2-M_Compensation[j].Encoder)*(M_Compensation[j+1].RightBottom-M_Compensation[j].RightBottom))
							/(M_Compensation[j+1].Encoder-M_Compensation[j].Encoder))+M_Compensation[j].RightBottom;
					M_CompensationNumber:=j;
					InitCompensationDatasDone:=TRUE;
				ELSIF j=18 AND UserRightGapPositionNew/2=M_Compensation[i].Encoder THEN		(*Gap=14µÄÌØÊâÇé¿ö*)
					(**)
					RightTopLinPositionNew:=M_Compensation[i].RightTop;
					RightBottomLinPositionNew:=M_Compensation[i].RightBottom;
					M_CompensationNumber:=j;
					InitCompensationDatasDone:=TRUE;
				ELSE
					RightTopLinPositionNew:=UserGapPositionNew/2;
					RightBottomLinPositionNew:=UserGapPositionNew/2;
					M_CompensationNumber:=j;
					InitCompensationDatasDone:=TRUE;
				END_IF
			END_IF
		END_FOR
		//
		//2.不论taper还是非taper模式，左轴gap都有左轴发推算，右轴gap由右轴反推算。taper为右gap-左gap
		//
		//左轴显示位置反结算
		FOR k:= 1 TO 17 DO
				IF Pos_LeftTopLin<M_Compensation[k+1].LeftTop AND Pos_LeftTopLin>=M_Compensation[k].LeftTop THEN
					UserGapPositionDisplay_FromLeftTop:=2*(((Pos_LeftTopLin-M_Compensation[k].LeftTop)*(M_Compensation[k+1].Encoder-M_Compensation[k].Encoder))
												/(M_Compensation[k+1].LeftTop-M_Compensation[k].LeftTop)+M_Compensation[k].Encoder);
					UserGapPositionDisplay_FromLeftBottom:=2*(((Pos_LeftBottomLin-M_Compensation[k].LeftBottom)*(M_Compensation[k+1].Encoder-M_Compensation[k].Encoder))
												/(M_Compensation[k+1].LeftBottom-M_Compensation[k].LeftBottom)+M_Compensation[k].Encoder);
					UserGapPositionDisplay:=DINT_TO_LREAL(LREAL_TO_DINT(((UserGapPositionDisplay_FromLeftTop+UserGapPositionDisplay_FromLeftBottom)/2)*100000))/100000;
				END_IF
		END_FOR
		//右轴显示位置反结算
		FOR m:= 1 TO 17 DO
				IF Pos_RightTopLin<M_Compensation[m+1].RightTop AND Pos_RightTopLin>=M_Compensation[m].RightTop THEN
					UserRightGapPositionDisplay_FromRightTop:=2*(((Pos_RightTopLin-M_Compensation[m].RightTop)*(M_Compensation[m+1].Encoder-M_Compensation[m].Encoder))
												/(M_Compensation[m+1].RightTop-M_Compensation[m].RightTop)+M_Compensation[m].Encoder);
					UserRightGapPositionDisplay_FromRightBottom:=2*(((Pos_RightBottomLin-M_Compensation[m].RightBottom)*(M_Compensation[m+1].Encoder-M_Compensation[m].Encoder))
												/(M_Compensation[m+1].RightBottom-M_Compensation[m].RightBottom)+M_Compensation[m].Encoder);
					UserRightGapPositionDisplay:=(UserRightGapPositionDisplay_FromRightTop+UserRightGapPositionDisplay_FromRightBottom)/2;
				END_IF
		END_FOR
		IF TaperOrNot OR (Global_ChainProtection_MPS_Triggered OR Global_ChainProtection_EPS_Triggered)  THEN//安全联锁触发时，需要UserTaperPositionDisplay作为A_MonitoringAllAxis的保护
			UserTaperPositionDisplay:=DINT_TO_LREAL(LREAL_TO_DINT((UserRightGapPositionDisplay-UserGapPositionDisplay)*100000))/100000;
			UserTaperVelocityDisplay:=DINT_TO_LREAL(LREAL_TO_DINT((Velo_RightTopLin+Velo_RightBottomLin)*100000))/100000;
		END_IF
		
		UserTaperPositionDisplayBLSide:=DINT_TO_LREAL(LREAL_TO_DINT((UserTaperPositionDisplay/IDTaperAndBLTaperScale*100000)))/100000;
		
		(*速度可以不用解算，直接用即可*)
		LeftTopLinVelocityDisplay:=Velo_LeftTopLin;
		RightTopLinVelocityDisplay:=Velo_RightTopLin;
		LeftBottomLinVelocityDisplay:=Velo_LeftBottomLin;
		RightBottomLinVelocityDisplay:=Velo_RightBottomLin;
		//Gap velocity
		UserGapVelocityDisplay:=DINT_TO_LREAL(LREAL_TO_DINT(((LeftTopLinVelocityDisplay+RightTopLinVelocityDisplay+
			LeftBottomLinVelocityDisplay+RightBottomLinVelocityDisplay)/2)*100000))/100000;
	
			(*解算单轴位置后，核验并做保护*)
		IF ABS(LeftTopLinPositionNew-UserGapPositionNew/2)>Threshold_motorsTargetPosCalculate THEN
			ErrorID:=1601;
			Error:=TRUE;
			ErrorDescription:='LeftTop Threshold_motorsTargetPosCalculate';
			FB_PlcEmergencyStop();
		END_IF
		//注意右轴解算以UserRightGapPositionNew为基准，考虑到taper
		IF ABS(RightTopLinPositionNew-UserRightGapPositionNew/2)>Threshold_motorsTargetPosCalculate THEN
			ErrorID:=1602;
			Error:=TRUE;
			ErrorDescription:='RightTop Threshold_motorsTargetPosCalculate';
			FB_PlcEmergencyStop();
		END_IF
		IF ABS(LeftBottomLinPositionNew-UserGapPositionNew/2)>Threshold_motorsTargetPosCalculate THEN
			ErrorID:=1603;
			Error:=TRUE;
			ErrorDescription:='LeftBottom Threshold_motorsTargetPosCalculate';
			FB_PlcEmergencyStop();
		END_IF
		//注意右轴解算以UserRightGapPositionNew为基准，考虑到taper
		IF ABS(RightBottomLinPositionNew-UserRightGapPositionNew/2)>Threshold_motorsTargetPosCalculate THEN
			ErrorID:=1604;
			Error:=TRUE;
			ErrorDescription:='RightBottom Threshold_motorsTargetPosCalculate';
			FB_PlcEmergencyStop();
		END_IF
	END_IF
		

(*线站taper模式下，出入口电机位置都解算*)
	IF BLTaperMode THEN
		//
		//1.目标位置解算
		//
		(*通过补偿表解算四轴目标位置*)
		//左轴目标位置解算
		IF NOT BLTaperOrNot THEN
			BLUserTaperPositionNew:=0;
		END_IF
		BLUserLeftGapPositionNew:=UserGapPositionNew-BLUserTaperPositionNew*IDTaperAndBLTaperScale/2;
		BLUserRightGapPositionNew:=UserGapPositionNew+BLUserTaperPositionNew*IDTaperAndBLTaperScale/2;
		//左轴目标位置解算
		FOR	i:= 1 TO 17 DO
				IF BLUserLeftGapPositionNew/2<M_Compensation[i+1].Encoder AND BLUserLeftGapPositionNew/2>=M_Compensation[i].Encoder THEN
					IF i<>18 THEN
						LeftTopLinPositionNew:=(((BLUserLeftGapPositionNew/2-M_Compensation[i].Encoder)*(M_Compensation[i+1].LeftTop-M_Compensation[i].LeftTop))
								/(M_Compensation[i+1].Encoder-M_Compensation[i].Encoder))+M_Compensation[i].LeftTop;
						LeftBottomLinPositionNew:=(((BLUserLeftGapPositionNew/2-M_Compensation[i].Encoder)*(M_Compensation[i+1].LeftBottom-M_Compensation[i].LeftBottom))
								/(M_Compensation[i+1].Encoder-M_Compensation[i].Encoder))+M_Compensation[i].LeftBottom;
						M_CompensationNumber:=i;
						InitCompensationDatasDone:=TRUE;
					ELSIF i=18 AND BLUserLeftGapPositionNew/2=M_Compensation[i].Encoder THEN		(*Gap=14µÄÌØÊâÇé¿ö*)
						(**)
						LeftTopLinPositionNew:=M_Compensation[i].LeftTop;
						LeftBottomLinPositionNew:=M_Compensation[i].LeftBottom;
						M_CompensationNumber:=i;
						InitCompensationDatasDone:=TRUE;
					ELSE
						LeftTopLinPositionNew:=BLUserLeftGapPositionNew/2;
						LeftBottomLinPositionNew:=BLUserLeftGapPositionNew/2;
						M_CompensationNumber:=i;
						InitCompensationDatasDone:=TRUE;
					END_IF
				END_IF
		END_FOR
		//右轴目标位置解算
		FOR	j:= 1 TO 17 DO
			IF BLUserRightGapPositionNew/2<M_Compensation[j+1].Encoder AND BLUserRightGapPositionNew/2>=M_Compensation[j].Encoder THEN
				IF j<>18 THEN
					RightTopLinPositionNew:=(((BLUserRightGapPositionNew/2-M_Compensation[j].Encoder)*(M_Compensation[j+1].RightTop-M_Compensation[j].RightTop))
							/(M_Compensation[j+1].Encoder-M_Compensation[j].Encoder))+M_Compensation[j].RightTop;
					RightBottomLinPositionNew:=(((BLUserRightGapPositionNew/2-M_Compensation[j].Encoder)*(M_Compensation[j+1].RightBottom-M_Compensation[j].RightBottom))
							/(M_Compensation[j+1].Encoder-M_Compensation[j].Encoder))+M_Compensation[j].RightBottom;
					M_CompensationNumber:=j;
					InitCompensationDatasDone:=TRUE;
				ELSIF j=18 AND BLUserRightGapPositionNew/2=M_Compensation[i].Encoder THEN		(*Gap=14µÄÌØÊâÇé¿ö*)
					(**)
					RightTopLinPositionNew:=M_Compensation[i].RightTop;
					RightBottomLinPositionNew:=M_Compensation[i].RightBottom;
					M_CompensationNumber:=j;
					InitCompensationDatasDone:=TRUE;
				ELSE
					RightTopLinPositionNew:=UserGapPositionNew/2;
					RightBottomLinPositionNew:=UserGapPositionNew/2;
					M_CompensationNumber:=j;
					InitCompensationDatasDone:=TRUE;
				END_IF
			END_IF
		END_FOR
		//
		//2.不论taper还是非taper模式，左轴gap都有左轴发推算，右轴gap由右轴反推算。
		//
		//左轴显示位置反结算
		FOR k:= 1 TO 17 DO
				IF Pos_LeftTopLin<M_Compensation[k+1].LeftTop AND Pos_LeftTopLin>=M_Compensation[k].LeftTop THEN
					BLUserGapPositionDisplay_FromLeftTop:=2*(((Pos_LeftTopLin-M_Compensation[k].LeftTop)*(M_Compensation[k+1].Encoder-M_Compensation[k].Encoder))
												/(M_Compensation[k+1].LeftTop-M_Compensation[k].LeftTop)+M_Compensation[k].Encoder);
					BLUserGapPositionDisplay_FromLeftBottom:=2*(((Pos_LeftBottomLin-M_Compensation[k].LeftBottom)*(M_Compensation[k+1].Encoder-M_Compensation[k].Encoder))
												/(M_Compensation[k+1].LeftBottom-M_Compensation[k].LeftBottom)+M_Compensation[k].Encoder);
					BLUserLeftGapPositionDisplay:=DINT_TO_LREAL(LREAL_TO_DINT(((BLUserGapPositionDisplay_FromLeftTop+BLUserGapPositionDisplay_FromLeftBottom)/2)*100000))/100000;
				END_IF
		END_FOR
		//右轴显示位置反结算
		FOR m:= 1 TO 17 DO
				IF Pos_RightTopLin<M_Compensation[m+1].RightTop AND Pos_RightTopLin>=M_Compensation[m].RightTop THEN
					BLUserRightGapPositionDisplay_FromRightTop:=2*(((Pos_RightTopLin-M_Compensation[m].RightTop)*(M_Compensation[m+1].Encoder-M_Compensation[m].Encoder))
												/(M_Compensation[m+1].RightTop-M_Compensation[m].RightTop)+M_Compensation[m].Encoder);
					BLUserRightGapPositionDisplay_FromRightBottom:=2*(((Pos_RightBottomLin-M_Compensation[m].RightBottom)*(M_Compensation[m+1].Encoder-M_Compensation[m].Encoder))
												/(M_Compensation[m+1].RightBottom-M_Compensation[m].RightBottom)+M_Compensation[m].Encoder);
					BLUserRightGapPositionDisplay:=(BLUserRightGapPositionDisplay_FromRightTop+BLUserRightGapPositionDisplay_FromRightBottom)/2;
				END_IF
		END_FOR
		//IF TaperOrNot OR (Global_ChainProtection_MPS_Triggered OR Global_ChainProtection_EPS_Triggered)  THEN//安全联锁触发时，需要UserTaperPositionDisplay作为A_MonitoringAllAxis的保护
		//	UserTaperPositionDisplay:=DINT_TO_LREAL(LREAL_TO_DINT((UserRightGapPositionDisplay-UserGapPositionDisplay)/IDTaperAndBLTaperScale*100000))/100000;
		//	UserTaperVelocityDisplay:=DINT_TO_LREAL(LREAL_TO_DINT((Velo_RightTopLin+Velo_RightBottomLin)/IDTaperAndBLTaperScale/2*100000))/100000;
		//END_IF
		//位置反解算
		UserGapPositionDisplay:=DINT_TO_LREAL(LREAL_TO_DINT(((BLUserLeftGapPositionDisplay+BLUserRightGapPositionDisplay)/2)*100000))/100000;
		BLUserTaperPositionDisplay:=DINT_TO_LREAL(LREAL_TO_DINT(((BLUserRightGapPositionDisplay-BLUserLeftGapPositionDisplay)/IDTaperAndBLTaperScale)*100000))/100000;
		//速度反解算
		LeftTopLinVelocityDisplay:=Velo_LeftTopLin/IDTaperAndBLTaperScale;
		RightTopLinVelocityDisplay:=Velo_RightTopLin/IDTaperAndBLTaperScale;
		LeftBottomLinVelocityDisplay:=Velo_LeftBottomLin/IDTaperAndBLTaperScale;
		RightBottomLinVelocityDisplay:=Velo_RightBottomLin/IDTaperAndBLTaperScale;
		BLUserTaperVelocityDisplay:=DINT_TO_LREAL(LREAL_TO_DINT((RightTopLinVelocityDisplay+RightBottomLinVelocityDisplay-
								(LeftTopLinVelocityDisplay+LeftBottomLinVelocityDisplay))*100000))/100000;
	END_IF

END_IF
END_ACTION

ACTION A_MonitoringAllAxis:
(****************************************************************
NAME:			A_MonitoringAllAxis
DATA:			2018.1.9
VERSION:		1.0.0
DESCRIPTION:	

HISTORY:
				2017.1.9		NEW

***************************************************************)
IF  st_Power<>0 THEN
CASE moni_State OF
0:
		//
		//step1:根据四轴光栅，计算实际位置差和速度差
		//
		(*Top*)
		Diff_UserTopPos_actual:=ABS(Pos_leftTopLin-Pos_RightTopLin);
		(*Bottom*)
		Diff_UserBottomPos_actual:=ABS(Pos_LeftBottomLin-Pos_RightBottomLin);
		(*Left*)
		Diff_UserLeftPos_actual:=ABS(Pos_LeftTopLin-Pos_LeftBottomLin);
		(*Right*)
		Diff_UserRightPos_actual:=ABS(Pos_RightTopLin-Pos_RightBottomLin);
		(*Velocity*)
		(*Top*)
		Diff_UserTopVelo_actual:=ABS(Velo_leftTopLin-Velo_RightTopLin);
		(*Bottom*)
		Diff_UserBottomVelo_actual:=ABS(Velo_LeftBottomLin-Velo_RightBottomLin);
		(*Left*)
		Diff_UserLeftVelo_actual:=ABS(Velo_LeftTopLin-Velo_LeftBottomLin);
		(*Right*)
		Diff_UserRightVelo_actual:=ABS(Velo_RightTopLin-Velo_RightBottomLin);
		//
		//step2:分类计算阈值
		//
		//正常gap模式
		IF NormalGapMode THEN
			Threshold_UserTopPos_PLC:=Threshold_UserTopPos;//位置差=固有阈值，在参数表中调节
			Threshold_UserTopVelo_PLC:=Threshold_UserTopVelo+ABS(UserGapVelocityDisplay);//速度差=固有阈值+当前速度。因为有一轴停止，其它轴还在运动的情况
			Threshold_UserBottomPos_PLC:=Threshold_UserBottomPos;
			Threshold_UserBottomVelo_PLC:=Threshold_UserBottomVelo+ABS(UserGapVelocityDisplay);
			Threshold_UserLeftPos_PLC:=Threshold_UserLeftPos;
			Threshold_UserLeftVelo_PLC:=Threshold_UserLeftVelo+ABS(UserGapVelocityDisplay);
			Threshold_UserRightPos_PLC:=Threshold_UserRightPos;
			Threshold_UserRightVelo_PLC:=Threshold_UserRightVelo+ABS(UserGapVelocityDisplay);
		END_IF		
		//IDTaper模式
		IF IDTaperMode THEN
			Threshold_UserTopPos_PLC:=Threshold_UserTopPos+ABS(UserTaperPositionDisplay*1.1/2);//位置差=固有阈值+当前taper值的一半，1.1为安全系数
			Threshold_UserTopVelo_PLC:=Threshold_UserTopVelo+ABS(UserTaperVelocityDisplay*1.1/2);
			Threshold_UserBottomPos_PLC:=Threshold_UserBottomPos+ABS(UserTaperPositionDisplay*1.1/2);
			Threshold_UserBottomVelo_PLC:=Threshold_UserBottomVelo+ABS(UserTaperVelocityDisplay*1.1/2);
			Threshold_UserLeftPos_PLC:=Threshold_UserLeftPos+ABS(UserTaperPositionDisplay*1.1/2);
			Threshold_UserLeftVelo_PLC:=Threshold_UserLeftVelo+ABS(UserTaperVelocityDisplay*1.1/2);
			Threshold_UserRightPos_PLC:=Threshold_UserRightPos+ABS(UserTaperPositionDisplay*1.1/2);
			Threshold_UserRightVelo_PLC:=Threshold_UserRightVelo+ABS(UserTaperVelocityDisplay*1.1/2);
		END_IF
		//线站taper模式
		IF BLTaperMode THEN
			Threshold_UserTopPos_PLC:=Threshold_UserTopPos+ABS(BLUserTaperPositionDisplay*IDTaperAndBLTaperScale*1.1/2);//Top位置误差=gap运动细微误差+目标taper位置
			Threshold_UserTopVelo_PLC:=Threshold_UserTopVelo+ABS(BLUserTaperVelocityDisplay*IDTaperAndBLTaperScale*1.1/2);//Top速度误差=gap运动细微误差+gap目标速度。因为可能出现一个轴运动完了，另一个轴还在运动的情况
			Threshold_UserBottomPos_PLC:=Threshold_UserBottomPos+ABS(BLUserTaperPositionDisplay*IDTaperAndBLTaperScale*1.1/2);//Bottom同上
			Threshold_UserBottomVelo_PLC:=Threshold_UserBottomVelo+ABS(BLUserTaperVelocityDisplay*IDTaperAndBLTaperScale*1.1/2);
			Threshold_UserLeftPos_PLC:=Threshold_UserLeftPos+ABS(BLUserTaperPositionDisplay*IDTaperAndBLTaperScale*1.1/2);
			Threshold_UserLeftVelo_PLC:=Threshold_UserLeftVelo+ABS(BLUserTaperVelocityDisplay*IDTaperAndBLTaperScale*1.1/2);
			Threshold_UserRightPos_PLC:=Threshold_UserRightPos+ABS(BLUserTaperPositionDisplay*IDTaperAndBLTaperScale*1.1/2);
			Threshold_UserRightVelo_PLC:=Threshold_UserRightVelo+ABS(BLUserTaperVelocityDisplay*IDTaperAndBLTaperScale*1.1/2);
		END_IF
		//
		//step3:保护
		//
		IF Diff_UserTopPos_actual >Threshold_UserTopPos_PLC  THEN
				Error:=TRUE;
				ErrorID:=601;
				ErrorDescription:='Diff_UserTopPos_actual >Threshold_UserTopPos_PLC';
				moni_State:=-100;
		END_IF
		IF Diff_UserTopVelo_actual>Threshold_UserTopVelo_PLC  THEN
				Error:=TRUE;
				ErrorID:=602;
				ErrorDescription:='Diff_UserTopVelo_actual>Threshold_UserTopVelo_PLC';
				moni_State:=-100;
		END_IF
		IF Diff_UserBottomPos_actual>Threshold_UserBottomPos_PLC  THEN
				Error:=TRUE;
				ErrorID:=603;
				ErrorDescription:='Diff_UserBottomPos_actual>Threshold_UserBottomPos_PLC';
				moni_State:=-100;
		END_IF
		IF Diff_UserBottomVelo_actual>Threshold_UserBottomVelo_PLC  THEN
				Error:=TRUE;
				ErrorID:=604;
				ErrorDescription:='Diff_UserBottomVelo_actual>Threshold_UserBottomVelo_PLC';
				moni_State:=-100;
		END_IF
		IF Diff_UserLeftPos_actual>Threshold_UserLeftPos_PLC  THEN
				Error:=TRUE;
				ErrorID:=605;
				ErrorDescription:='Diff_UserLeftPos_actual>Threshold_UserLeftPos_PLC';
				moni_State:=-100;
		END_IF
		IF  Diff_UserLeftVelo_actual>Threshold_UserLeftVelo_PLC THEN
				Error:=TRUE;
				ErrorID:=606;
				ErrorDescription:='Diff_UserLeftVelo_actual>Threshold_UserLeftVelo_PLC';
				moni_State:=-100;	
		END_IF
		IF Diff_UserRightPos_actual>Threshold_UserRightPos_PLC  THEN
				Error:=TRUE;
				ErrorID:=607;
				ErrorDescription:='Diff_UserRightPos_actual>Threshold_UserRightPos_PLC';
				moni_State:=-100;	
		END_IF
		IF  Diff_UserRightVelo_actual>Threshold_UserRightVelo_PLC THEN
				Error:=TRUE;
				ErrorID:=608;
				ErrorDescription:='Diff_UserRightVelo_actual>Threshold_UserRightVelo_PLC';
				moni_State:=-100;
		END_IF
		//单独拿出最大taper来做冗余保护
		IF IDTaperMode THEN
			IF  Diff_UserTopPos_actual > max_UserTaperPositionNew*1.1/2 THEN
					Error:=TRUE;
					ErrorID:=609;
					ErrorDescription:='Diff_UserTopPos_actual > max_UserTaperPositionNew*1.1/2';
					moni_State:=-100;
			END_IF
			IF  Diff_UserBottomPos_actual > max_UserTaperPositionNew*1.1/2 THEN
					Error:=TRUE;
					ErrorID:=610;
					ErrorDescription:='Diff_UserBottomPos_actual > max_UserTaperPositionNew*1.1/2';
					moni_State:=-100;
			END_IF
		END_IF
		IF BLTaperMode THEN
			IF  Diff_UserTopPos_actual > (max_BLUserTaperPositionNew*IDTaperAndBLTaperScale+HysteresisError)*1.1/2 THEN//
					Error:=TRUE;
					ErrorID:=609;
					ErrorDescription:='Diff_UserTopPos_actual > (max_BLUserTaperPositionNew*IDTaperAndBLTaperScale+HysteresisError)*1.1/2';
					moni_State:=-100;
			END_IF
			IF  Diff_UserBottomPos_actual > (max_BLUserTaperPositionNew*IDTaperAndBLTaperScale+HysteresisError)*1.1/2 THEN//
					Error:=TRUE;
					ErrorID:=610;
					ErrorDescription:='Diff_UserBottomPos_actual > (max_BLUserTaperPositionNew*IDTaperAndBLTaperScale+HysteresisError)*1.1/2';
					moni_State:=-100;
			END_IF
		END_IF
-100:
		btn_UserGapStop:=TRUE;
		FB_PlcEmergencyStop();
		Error:=TRUE;
		LED_Error:=TRUE;
END_CASE
END_IF
END_ACTION

ACTION A_OneKeyToMaxGap:
//0.上升沿触发
//1.判断电机是否在开启状态,没有就打开电源
//2.判断是否在Moving状态,若有就Stop
//3.将磁间隙打开到至最大阈值
//4.到位后给出反馈
OneKeyToMaxGap_RTRIG(CLK:=btn_OneKeyToMaxGap);
IF OneKeyToMaxGap_RTRIG.Q THEN
	OneKeyToMaxGap_Triggered:=TRUE;
	OneKeyToMaxGap_Done:=FALSE;
END_IF
IF OneKeyToMaxGap_Triggered THEN
	CASE OneKeyToMaxGap_State OF
		0://1.判断电机是否在开启状态,没有就打开电源
			IF st_Power=1 THEN
				OneKeyToMaxGap_State:=1;
			ELSE
				btn_PowerOn:=TRUE;
				IF btn_PowerOn THEN
					A_PowerOn();
				END_IF
			END_IF
		1://1.判断是否在谱学扫描模式，如果是，则切换回正常运动模式
			IF IsSSMotionMode THEN
				SS_Stop:=TRUE;
				IsSSMotionMode:=FALSE;
			END_IF
			OneKeyToMaxGap_State:=2;
		2://判断是否在taper，如果在taper,则判断是否在运动，如果是，则停止运动,0.5sh后，转入下一步
			IF TaperOrNot THEN
				IF moveStatusLeftTop OR moveStatusRightTop OR moveStatusLeftBottom OR moveStatusRightBottom THEN
					btn_UserGapStop:=TRUE;
				ELSE
					OneKeyToMaxGap_TON_Stop2Move_InTaperMode(PT:=T#0.5S);
					OneKeyToMaxGap_TON_Stop2Move_InTaperMode.IN:=TRUE;
					IF OneKeyToMaxGap_TON_Stop2Move_InTaperMode.Q THEN
						TaperOrNot:=FALSE;//关闭taper模式
						OneKeyToMaxGap_State:=3;
						OneKeyToMaxGap_TON_Stop2Move_InTaperMode.IN:=FALSE;
					END_IF
				END_IF
			ELSE
				OneKeyToMaxGap_State:=3;
			END_IF
		3://3.判断是否在Moving状态,若有就Stop.Taper模式已处理完，此处开始走正常GAP开合逻辑
			IF moveStatusLeftTop OR moveStatusRightTop OR moveStatusLeftBottom OR moveStatusRightBottom THEN
				btn_UserGapStop:=TRUE;
			ELSE
				OneKeyToMaxGap_TON_Stop2Move(PT:=T#0.5S);
				OneKeyToMaxGap_TON_Stop2Move.IN:=TRUE;
				IF OneKeyToMaxGap_TON_Stop2Move.Q THEN
					OneKeyToMaxGap_State:=4;
					OneKeyToMaxGap_TON_Stop2Move.IN:=FALSE;
				END_IF
			END_IF
		4://4.将磁间隙打开到至最大阈值
			OneKeyToMaxGap_TON(PT:=INT_TO_TIME(LREAL_TO_INT(max_UserGapPositionNew+30))*1000);
			OneKeyToMaxGap_TON.IN:=TRUE;
			OneKeyToMaxGap_TON_Power2Move(PT:=T#0.1S);
			OneKeyToMaxGap_TON_Power2Move.IN:=TRUE;
			UserGapPositionNew:=max_UserGapPositionNew;
			UserGapVelocityNew:=1;
			btn_UserGapMove:=TRUE;
			IF OneKeyToMaxGap_TON_Power2Move.Q THEN
				OneKeyToMaxGap_TON_Power2Move.IN:=FALSE;
				IF FB_MOVE.BCGapDone THEN
					OneKeyToMaxGap_State:=88;
				END_IF
			END_IF
			IF OneKeyToMaxGap_TON.Q THEN//如果150s后，还没有运动到指定gap，则报错
				OneKeyToMaxGap_TON.IN:=FALSE;
				OneKeyToMaxGap_State:=-100;
			END_IF
			IF  btn_UserGapStop THEN
				//
				OneKeyToMaxGap_State:=0;
				OneKeyToMaxGap_Triggered:=FALSE;
				btn_OneKeyToMaxGap:=FALSE;
				OneKeyToMaxGap_Triggered:=FALSE;
				OneKeyToMaxGap_State:=0;
			END_IF
		88://6.到位后给出反馈
			OneKeyToMaxGap_Done:=TRUE;	
			Error:=FALSE;
			ErrorID:=0;
			ErrorDescription:='';
			btn_OneKeyToMaxGap:=FALSE;
			OneKeyToMaxGap_Triggered:=FALSE;
			OneKeyToMaxGap_State:=0;
				
		-100:
			OneKeyToMaxGap_Done:=FALSE;
			Error:=TRUE;
			ErrorID:=1705;
			ErrorDescription:='OneKeyToMaxGap Fail';
			btn_OneKeyToMaxGap:=FALSE;
			OneKeyToMaxGap_Triggered:=FALSE;
			OneKeyToMaxGap_State:=0;
	END_CASE
END_IF
END_ACTION

ACTION A_OneKeyToTaperZero:
IF NormalGapMode THEN
	RETURN;
END_IF
//0.上升沿触发
//1.判断当前taper功能是否开启，没有则RETURN
//2.taper=0，目标gap=当前gap,调用btn_GapMove，运动完成
//3.taperOrNot关闭

//0.上升沿触发
OneKeyToTaperZero_RTRIG(CLK:=btn_OneKeyToTaperZero);
IF OneKeyToTaperZero_RTRIG.Q THEN
	OneKeyToTaperZero_Triggered:=TRUE;
	OneKeyToTaperZero_Done:=FALSE;
END_IF
IF IDTaperMode AND UserTaperVelocityNew<>0 THEN
	OneKeyToTaperZero_TON(PT:=INT_TO_TIME(LREAL_TO_INT((CurrentTaperInit+HysteresisError*10)/UserTaperVelocityNew))*1000);
END_IF
IF BLTaperMode AND BLUserTaperVelocityNew<>0 THEN
	OneKeyToTaperZero_TON(PT:=INT_TO_TIME(LREAL_TO_INT((CurrentTaperInit+HysteresisError*20)/BLUserTaperVelocityNew))*1000);
END_IF
OneKeyToTaperZero_Delay(PT:=T#0.5S);
IF OneKeyToTaperZero_Triggered THEN
	CASE OneKeyToTaperZero_State OF
		0://1.判断当前taper功能是否开启，没有则RETURN
			IF IDTaperMode OR BLTaperMode THEN
				OneKeyToTaperZero_State:=1;
			END_IF
		1://2.taper=0，目标gap=当前gap,调用btn_GapMove
			IF IDTaperMode THEN
				UserGapPositionNew:=UserGapPositionDisplay;
				UserTaperPositionNew:=0;
				btn_UserGapMove:=TRUE;
				OneKeyToTaperZero_State:=2;
				IF UserTaperPositionDisplay<=Threshold_TaperChangeFlag THEN//本来当前taper就基本是0,直接关闭taper功能即可
					OneKeyToTaperZero_State:=3;
				END_IF
				CurrentTaperInit:=UserTaperPositionDisplay;
			END_IF
			IF BLTaperMode THEN
				UserGapPositionNew:=UserGapPositionDisplay;
				BLUserTaperPositionNew:=0;
				btn_UserGapMove:=TRUE;
				OneKeyToTaperZero_State:=2;
				IF BLUserTaperPositionDisplay<=Threshold_TaperChangeFlag THEN//本来当前taper就基本是0,直接关闭taper功能即可
					OneKeyToTaperZero_State:=3;
				END_IF
				CurrentTaperInit:=BLUserTaperPositionDisplay;
			END_IF
		2://Move
			OneKeyToTaperZero_TON.IN:=TRUE;
			IF NOT OneKeyToTaperZero_TON.Q THEN
				IF n_state=88 THEN//运动完成
					OneKeyToTaperZero_State:=3;
				END_IF
			ELSE//时间到，还没有运动完，报错
				OneKeyToTaperZero_TON.IN:=FALSE;
				OneKeyToTaperZero_State:=-100;
			END_IF
		3://taper功能关闭
			//延迟0.5s后关闭
			OneKeyToTaperZero_Delay.IN:=TRUE;
			IF OneKeyToTaperZero_Delay.Q THEN
				IF IDTaperMode THEN
					TaperOrNot:=FALSE;
				END_IF
				IF BLTaperMode THEN
					BLTaperOrNot:=FALSE;
				END_IF
				OneKeyToTaperZero_State:=88;				
				OneKeyToTaperZero_Delay.IN:=FALSE;
			END_IF
		88://到位
			OneKeyToTaperZero_Done:=TRUE;	
			Error:=FALSE;
			ErrorID:=0;
			ErrorDescription:='';
			btn_OneKeyToTaperZero:=FALSE;
			OneKeyToTaperZero_Triggered:=FALSE;
			OneKeyToTaperZero_State:=0;
			OneKeyToTaperZero_TON.IN:=FALSE;
			OneKeyToTaperZero_Delay.IN:=FALSE;				
		-100:
			OneKeyToTaperZero_Done:=FALSE;
			Error:=TRUE;
			ErrorID:=1705;
			ErrorDescription:='OneKeyToTaperZero Fail';
			btn_OneKeyToTaperZero:=FALSE;
			OneKeyToTaperZero_Triggered:=FALSE;
			OneKeyToTaperZero_State:=0;
			OneKeyToTaperZero_TON.IN:=FALSE;
	END_CASE
END_IF
END_ACTION

ACTION A_PowerOff:
CASE d_state OF
		0:(*PowerOff*)
			FB_Power(Off:=TRUE);
				d_state:=1;
		1:
			IF NOT FB_power.OffStatus THEN
				d_state:=1;
			ELSE
				d_state:=88;
			END_IF
		88:(*ResetAllState*)
			btn_PowerOn:=FALSE;
			btn_UserGapMove:=FALSE;
			btn_UserGapStop:=FALSE;
			LeftTopLinMoveIndicator:=0;
			RightTopLinMoveIndicator:=0;
			LeftBottomLinMoveIndicator:=0;
			RightBottomLinMoveIndicator:=0;
			fb_ton1.IN:=FALSE;
			fb_ton2.IN:=FALSE;
			fb_ton3.IN:=FALSE;
			State:=0;
			Busy:=FALSE;
			InitPowerDone:=FALSE;
			InitCompensationDatasDone:=FALSE;
			Error:=FALSE;
			ErrorID:=0;
			m_state:=0;
			n_state:=0;
			s_state:=0;
			btn_PowerOff:=FALSE;
			d_state:=0;
			Led_Run:=FALSE;
			Led_Error:=FALSE;
			moni_State:=0;
			i:=0;
END_CASE
END_ACTION

ACTION A_PowerOn:
(****************************************************************
NAME:			A_PowerOn
DATA:			2018.1.9
VERSION:		1.0.0
DESCRIPTION:	

HISTORY:
				2019.1.9		NEW

***************************************************************)
fb_ton3(PT:=t#0.5s);
CASE State OF
	0:	(*FB_Power_On*)
		FB_Power(On:=TRUE);
		fb_ton3.IN:=TRUE;
		State:=1;
	1:	(*wait*)
		FB_power();
		IF NOT FB_power.OnStatus THEN
			IF NOT fb_ton3.Q THEN
				State:=1;
			ELSE
				ErrorID:=1;
				State:=99;
			END_IF
		ELSE
			State:=88;
		END_IF
	88:	(*All Done*)
		btn_PowerOn:=FALSE;
		State:=0;
		Error:=FALSE;
		ErrorID:=0;
		Busy:=FALSE;
		InitPowerDone:=TRUE;
		FB_power.On:=FALSE;
		fb_ton3.IN:=FALSE;
		LED_Error:=FALSE;
	99:
		Error:=TRUE;
		//ErrorID:=701;
		//ErrorDescription:='power on error';		
		btn_PowerOn:=FALSE;
		State:=99;
		Busy:=FALSE;
		InitPowerDone:=FALSE;
		fb_ton3.IN:=FALSE;
		LED_Error:=TRUE;
END_CASE
END_ACTION

ACTION A_RegularMotion:
//Taper运动保护
A_TaperMotionProtection();

(*分别比较四轴目标位置与当前位置的差，如果目标位置比当前位置低，则需要运动到更低-回程差一半；再运动至最终目标位置*)
//只在m=和n=0的时候判断，否则会出现一些BUG，比如往大间隙开时，运动到位后m不能回到0.
IF m_state=0 AND n_state=0 THEN
		TargetPosLessThanCurrentPos:=FALSE;
	IF LeftTopLinPositionNew-Pos_LeftTopLin<-LEDriftErrorThreshold THEN
			TargetPosLessThanCurrentPos:=TRUE;
			TargetLTPosLessThanCurrentLTPos:=TRUE;
	ELSE
				TargetLTPosLessThanCurrentLTPos:=FALSE;
	END_IF
	IF RightTopLinPositionNew-Pos_RightTopLin<-LEDriftErrorThreshold THEN
			TargetPosLessThanCurrentPos:=TRUE;
			TargetRTPosLessThanCurrentRTPos:=TRUE;
	ELSE
			TargetRTPosLessThanCurrentRTPos:=FALSE;
	END_IF
	IF LeftBottomLinPositionNew-Pos_LeftBottomLin<-LEDriftErrorThreshold THEN
			TargetPosLessThanCurrentPos:=TRUE;
			TargetLBPosLessThanCurrentLBPos:=TRUE;
	ELSE
			TargetLBPosLessThanCurrentLBPos:=FALSE;
	END_IF
	IF RightBottomLinPositionNew-Pos_RightBottomLin<-LEDriftErrorThreshold THEN
			TargetPosLessThanCurrentPos:=TRUE;
			TargetRBPosLessThanCurrentRBPos:=TRUE;
	ELSE
			TargetRBPosLessThanCurrentRBPos:=FALSE;
	END_IF
END_IF

(*Move*)
IF InitCompensationDatasDone THEN
		(*四轴目标位置都大于当前位置，直接走到目标位置即可，不需要先走到考虑回城误差的临时位置*)
		IF NOT TargetPosLessThanCurrentPos AND NOT HysteresisMoving THEN
			CASE m_state OF
				0:
					FB_Move.Mode:=5;						//1.gap;2.single;3.taper;4.debug;5.BCGap&UserMode
					FB_Move.CoupleState:=st_Couple;			
					FB_Move.PowerState:=st_Power;						
			
					IF btn_UserGapMove THEN
						IF NOT st_Power THEN
							ErrorID:=1501;
							Error:=TRUE;
							ErrorDescription:='Plz PowerOn Frist';
							LED_Error:=TRUE;
							//btn_UserGapMove:=FALSE;
							RETURN;
						ELSE
							ErrorID:=0;
							Error:=FALSE;
							ErrorDescription:='';
							LED_Error:=FALSE;
							//btn_UserGapMove:=TRUE;
						END_IF
						//目标位置赋值
						FB_Move.BCLeftTopPosition:=LeftTopLinPositionNew;
						FB_Move.BCRightTopPosition:=RightTopLinPositionNew;
						FB_Move.BCLeftBottomPosition:=LeftBottomLinPositionNew;
						FB_Move.BCRightBottomPosition:=RightBottomLinPositionNew;
						//目标速度赋值
						IF NormalGapMode THEN
							FB_Move.BCLeftTopVelocity:=UserGapVelocityNew/2;
							FB_Move.BCRightTopVelocity:=UserGapVelocityNew/2;
							FB_Move.BCLeftBottomVelocity:=UserGapVelocityNew/2;
							FB_Move.BCRightBottomVelocity:=UserGapVelocityNew/2;
						ELSIF IDTaperMode THEN
							FB_Move.BCLeftTopVelocity:=UserTaperVelocityNew/2;
							FB_Move.BCRightTopVelocity:=UserTaperVelocityNew/2;
							FB_Move.BCLeftBottomVelocity:=UserTaperVelocityNew/2;
							FB_Move.BCRightBottomVelocity:=UserTaperVelocityNew/2;
						ELSIF BLTaperMode THEN
							FB_Move.BCLeftTopVelocity:=BLUserTaperVelocityNew*IDTaperAndBLTaperScale/4;
							FB_Move.BCRightTopVelocity:=BLUserTaperVelocityNew*IDTaperAndBLTaperScale/4;
							FB_Move.BCLeftBottomVelocity:=BLUserTaperVelocityNew*IDTaperAndBLTaperScale/4;
							FB_Move.BCRightBottomVelocity:=BLUserTaperVelocityNew*IDTaperAndBLTaperScale/4;
						ELSE
							FB_Move.BCLeftTopVelocity:=0;
							FB_Move.BCRightTopVelocity:=0;
							FB_Move.BCLeftBottomVelocity:=0;
							FB_Move.BCRightBottomVelocity:=0;
						END_IF
						FB_Move.BCGapMove:=TRUE;
						m_state:=1;
						FB_Move();
					END_IF
				1:
					btn_UserGapMove:=FALSE;
					FB_Move();
					IF NOT FB_Move.BCGapDone THEN
						Led_Run:=TRUE;
						m_state:=1;
					ELSE
						m_state:=88;
					END_IF
				88:
					btn_UserGapMove:=FALSE;
					Led_Run:=FALSE;
					m_state:=0;
			END_CASE
		(*四轴有目标位置小于当前位置，先走到临时位置，再走到目标位置*)
		ELSE
			CASE n_state OF
				0:
					FB_Move.Mode:=5;						//1.gap;2.single;3.taper;4.debug;5.BCGap&UserMode;5:userMode_2
					FB_Move.CoupleState:=st_Couple;			
					FB_Move.PowerState:=st_Power;			
					IF btn_UserGapMove THEN	
						IF NOT st_Power THEN
							ErrorID:=1501;
							Error:=TRUE;
							ErrorDescription:='Plz PowerOn Frist';
							LED_Error:=TRUE;
							//btn_UserGapMove:=FALSE;
							RETURN;
						ELSE
							ErrorID:=0;
							Error:=FALSE;
							ErrorDescription:='';
							LED_Error:=FALSE;
							//btn_UserGapMove:=TRUE;
						END_IF						
						//
						IF TargetLTPosLessThanCurrentLTPos THEN			
							FB_Move.BCLeftTopPosition:=LeftTopLinPositionNew-HysteresisError/2;
						ELSE
							FB_Move.BCLeftTopPosition:=LeftTopLinPositionNew;	
						END_IF
						//
						IF TargetRTPosLessThanCurrentRTPos THEN 
							FB_Move.BCRightTopPosition:=RightTopLinPositionNew-HysteresisError/2;
						ELSE					
							FB_Move.BCRightTopPosition:=RightTopLinPositionNew;
						END_IF
						//
						IF TargetLBPosLessThanCurrentLBPos THEN
							FB_Move.BCLeftBottomPosition:=LeftBottomLinPositionNew-HysteresisError/2;
						ELSE
							FB_Move.BCLeftBottomPosition:=LeftBottomLinPositionNew;
						END_IF
						//
						IF TargetRBPosLessThanCurrentRBPos THEN
							FB_Move.BCRightBottomPosition:=RightBottomLinPositionNew-HysteresisError/2;
						ELSE
							FB_Move.BCRightBottomPosition:=RightBottomLinPositionNew;
						END_IF	
						//	close gap情况下，加入了LeftTopLinPositionNewTemp。//
						//如果在往小间隙运行过程中，改变了目标gap，会在第到达第一次目标位置后，继续向第二
						//次输入的目标运动，而不会回到第一次的目标位置。用temp锁定目标位置
						LeftTopLinPositionNewTemp:=LeftTopLinPositionNew;
						RightTopLinPositionNewTemp:=RightTopLinPositionNew;
						LeftBottomLinPositionNewTemp:=LeftBottomLinPositionNew;
						RightBottomLinPositionNewTemp:=RightBottomLinPositionNew;
			
						//
						IF NormalGapMode THEN
							FB_Move.BCLeftTopVelocity:=UserGapVelocityNew/2;
							FB_Move.BCRightTopVelocity:=UserGapVelocityNew/2;
							FB_Move.BCLeftBottomVelocity:=UserGapVelocityNew/2;
							FB_Move.BCRightBottomVelocity:=UserGapVelocityNew/2;
							IF UserGapVelocityNew >1 THEN								  
								ErrorID:=1502;
								Error:=TRUE;
								ErrorDescription:='UserGapVelocityNew must<=1';
								LED_Error:=TRUE;
								btn_UserGapMove:=FALSE;
								RETURN;
							ELSE
								ErrorID:=0;
								Error:=FALSE;
								ErrorDescription:='';
								LED_Error:=FALSE;	
							END_IF									
						ELSIF IDTaperMode THEN
							FB_Move.BCLeftTopVelocity:=UserTaperVelocityNew/2;
							FB_Move.BCRightTopVelocity:=UserTaperVelocityNew/2;
							FB_Move.BCLeftBottomVelocity:=UserTaperVelocityNew/2;
							FB_Move.BCRightBottomVelocity:=UserTaperVelocityNew/2;
						ELSIF BLTaperMode THEN
							FB_Move.BCLeftTopVelocity:=BLUserTaperVelocityNew*IDTaperAndBLTaperScale/4;
							FB_Move.BCRightTopVelocity:=BLUserTaperVelocityNew*IDTaperAndBLTaperScale/4;
							FB_Move.BCLeftBottomVelocity:=BLUserTaperVelocityNew*IDTaperAndBLTaperScale/4;
							FB_Move.BCRightBottomVelocity:=BLUserTaperVelocityNew*IDTaperAndBLTaperScale/4;
						ELSE
							FB_Move.BCLeftTopVelocity:=0;
							FB_Move.BCRightTopVelocity:=0;
							FB_Move.BCLeftBottomVelocity:=0;
							FB_Move.BCRightBottomVelocity:=0;
						END_IF	

						FB_Move.BCGapMove:=TRUE;
						FB_Move();
						HysteresisMoving:=TRUE;		
						n_state:=1;	
					END_IF
				1:
					btn_UserGapMove:=FALSE;
					FB_Move();
					IF NOT FB_Move.BCGapDone THEN			(*还未运动到位置,运动过程中*)
						Led_Run:=TRUE;
						n_state:=1;
					ELSE									
						n_state:=2;							(*转到下一步，运动到最终位置*)
						FB_Move.BCGapMove:=FALSE;
						//Led_Run:=FALSE;
					END_IF
				2:
					FB_Move.BCGapReset:=FALSE;
					FB_Move.Mode:=5;						//1.gap;2.single;3.taper;4.debug;5.BCGap&UserMode
					FB_Move.CoupleState:=st_Couple;			
					FB_Move.PowerState:=st_Power;			
					FB_Move.BCGapMove:=TRUE;
					//直接走到目标位置，已经走到位置的，可以继续下命令，只不过它不在走了而已
					FB_Move.BCLeftTopPosition:=LeftTopLinPositionNewTemp;	
					FB_Move.BCRightTopPosition:=RightTopLinPositionNewTemp;
					FB_Move.BCLeftBottomPosition:=LeftBottomLinPositionNewTemp;
					FB_Move.BCRightBottomPosition:=RightBottomLinPositionNewTemp;
					//
					//目标速度赋值
					IF NormalGapMode THEN
						FB_Move.BCLeftTopVelocity:=UserGapVelocityNew/2;
						FB_Move.BCRightTopVelocity:=UserGapVelocityNew/2;
						FB_Move.BCLeftBottomVelocity:=UserGapVelocityNew/2;
						FB_Move.BCRightBottomVelocity:=UserGapVelocityNew/2;
					ELSIF IDTaperMode THEN
						FB_Move.BCLeftTopVelocity:=UserTaperVelocityNew/2;
						FB_Move.BCRightTopVelocity:=UserTaperVelocityNew/2;
						FB_Move.BCLeftBottomVelocity:=UserTaperVelocityNew/2;
						FB_Move.BCRightBottomVelocity:=UserTaperVelocityNew/2;
					ELSIF BLTaperMode THEN
						FB_Move.BCLeftTopVelocity:=BLUserTaperVelocityNew*IDTaperAndBLTaperScale/4;
						FB_Move.BCRightTopVelocity:=BLUserTaperVelocityNew*IDTaperAndBLTaperScale/4;
						FB_Move.BCLeftBottomVelocity:=BLUserTaperVelocityNew*IDTaperAndBLTaperScale/4;
						FB_Move.BCRightBottomVelocity:=BLUserTaperVelocityNew*IDTaperAndBLTaperScale/4;
					ELSE
						FB_Move.BCLeftTopVelocity:=0;
						FB_Move.BCRightTopVelocity:=0;
						FB_Move.BCLeftBottomVelocity:=0;
						FB_Move.BCRightBottomVelocity:=0;
					END_IF
					FB_Move();							
					n_state:=3;
				3:
					FB_Move();
					IF NOT FB_Move.BCGapDone THEN			(*还未运动到位置,运动过程中*)
						Led_Run:=TRUE;
						n_state:=3;
					ELSE									
						n_state:=88;							(*运动到了最终位置*)
					END_IF
					(*
					IF NOT Unreach_LS_Bottom THEN
						n_state:=88;							(*在运动过程中如果碰到下限位，则也转到下一步，运动到最终位置*)
						FB_Move.BCGapMove_2:=FALSE;
					END_IF
					*)
				88:
					btn_UserGapMove:=FALSE;					
					Led_Run:=FALSE;
					n_state:=0;
					HysteresisMoving:=FALSE;
			END_CASE
		END_IF
	//
	//FB_Move.BCLeftTopPosition等四轴位置监控
	//
END_IF

IF btn_UserGapStop OR btn_Reset THEN
	FB_Move.BCGapReset:=TRUE;
	FB_Move();	
	btn_UserGapMove:=FALSE;	
	m_state:=0;	
	n_state:=0;	
	HysteresisMoving:=FALSE;
	CASE s_state OF
			0:
				FB_Stop.Mode:=5;	
				FB_Stop.CoupleState:=st_Couple;	
				FB_Stop.PowerState:=st_Power;
				FB_Stop.BCGapStop:=TRUE;
				FB_Stop();	
				s_state:=1;
			1:
				FB_Stop();
				IF NOT FB_Stop.BCGapDone THEN
					s_state:=1;
				ELSE
					s_state:=88;
				END_IF
			88:
				btn_UserGapStop:=FALSE;	
				FB_Move.BCGapReset:=FALSE;
				btn_reset:=FALSE;
				s_state:=0;
		END_CASE
END_IF

(*触发限位开关后，相当于点击了Stop按钮*)
FTrig_ReachLS(CLK:=Unreach_LS_Far AND Unreach_LS_Near);
IF FTrig_ReachLS.Q THEN
	btn_UserGapStop:=TRUE;
END_IF
END_ACTION

ACTION A_SpectroscopyScanningMotion:
(*输入保护*)
IF SS_Move AND SSMotionMode AND NOT RegularMotionMode THEN
	IF NOT inRange_SS_StepSize THEN
		SS_Stop:=TRUE;
		SS_Move:=FALSE;
		Error:=TRUE;
		ErrorId:=805;
		ErrorDescription:='target StepSize out of range,please check';
		RETURN;
	ELSE
		//SS_Stop:=FALSE;
		Error:=FALSE;
		ErrorId:=0;
		ErrorDescription:='';	
	END_IF
	//
	IF NOT inRange_SS_StepNumber THEN
		SS_Stop:=TRUE;
		SS_Move:=FALSE;
		Error:=TRUE;
		ErrorId:=806;
		ErrorDescription:='target StepNumber out of range,please check';
		RETURN;
	ELSE
		//SS_Stop:=FALSE;
		Error:=FALSE;
		ErrorId:=0;
		ErrorDescription:='';	
	END_IF
	IF NOT inRange_SS_StepVelocity THEN
		SS_Stop:=TRUE;
		SS_Move:=FALSE;
		Error:=TRUE;
		ErrorId:=807;
		ErrorDescription:='target StepVelocity out of range,please check';
		RETURN;
	ELSE
		//SS_Stop:=FALSE;
		Error:=FALSE;
		ErrorId:=0;
		ErrorDescription:='';	
	END_IF
	IF NOT inRange_StepEachTime_ms THEN
		SS_Stop:=TRUE;
		SS_Move:=FALSE;
		Error:=TRUE;
		ErrorId:=808;
		ErrorDescription:='target StepEachTime_ms out of range,please check';
		RETURN;
	ELSE
		//SS_Stop:=FALSE;
		Error:=FALSE;
		ErrorId:=0;
		ErrorDescription:='';	
	END_IF
END_IF
(*单步时长转换*)
StepEachTime:=INT_TO_TIME(StepEachTime_ms);
SS_TON(PT:=StepEachTime);
(*上升沿触发，初始SS位置=当前磁间隙*)
RTRG_SS_StartPositionDisplay(CLK:=SS_Move);
IF RTRG_SS_StartPositionDisplay.Q THEN
	SS_StartPositionDisplay:=UserGapPositionDisplay;
	SS_InitStartPositionDone:=TRUE;
END_IF
(*SS主程序*)
IF InitPowerDone AND InitCompensationDatasDone AND SS_Move AND SS_InitStartPositionDone THEN
	IF NOT st_Power THEN
		ErrorID:=1501;
		Error:=TRUE;
		ErrorDescription:='Plz PowerOn Frist';
		LED_Error:=TRUE;
		//btn_UserGapMove:=FALSE;
		RETURN;
	ELSE
		ErrorID:=0;
		Error:=FALSE;
		ErrorDescription:='';
		LED_Error:=FALSE;
		//btn_UserGapMove:=TRUE;
	END_IF	
CASE SS_MoveState OF
		0:
				//UserGapPositionNew:=UserGapPositionDisplay+SS_StepSize;
				UserGapPositionNew:=SS_StartPositionDisplay+SS_StepSize*(SS_currentStep+1);
				A_InitCompensationData();
				FB_Move.Mode:=5;						//1.gap;2.single;3.taper;4.debug;5.BCGap&UserMode
				FB_Move.CoupleState:=st_Couple;			
				FB_Move.PowerState:=st_Power;							
				FB_Move.BCLeftTopPosition:=LeftTopLinPositionNew;
				FB_Move.BCLeftTopVelocity:=SS_StepVelocity/2;
				FB_Move.BCRightTopPosition:=RightTopLinPositionNew;
				FB_Move.BCRightTopVelocity:=SS_StepVelocity/2;
				FB_Move.BCLeftBottomPosition:=LeftBottomLinPositionNew;
				FB_Move.BCLeftBottomVelocity:=SS_StepVelocity/2;
				FB_Move.BCRightBottomPosition:=RightBottomLinPositionNew;
				FB_Move.BCRightBottomVelocity:=SS_StepVelocity/2;		
				FB_Move.BCGapMove:=TRUE;
				FB_Move();
				SS_MoveState:=1;
		1:
				SS_TON.IN:=TRUE;
				FB_Move();
				IF FB_Move.GapMoving AND NOT SS_TimeCountBegin THEN
					SS_StepSystemTime_Begin[SS_currentStep]:=F_GetSysTime();
					SS_TimeCountBegin:=TRUE;
				END_IF
				IF NOT FB_Move.BCGapDone THEN			
					Led_Run:=TRUE;
					SS_MoveState:=1;
				ELSE									
					SS_MoveState:=66;
					SS_StepSystemTime_End[SS_currentStep]:=F_GetSysTime();
					SS_StepCountTime[SS_currentStep]:=SS_StepSystemTime_End[SS_currentStep]-SS_StepSystemTime_Begin[SS_currentStep];
					SS_TimeCountBegin:=FALSE;
				END_IF
		66:
				SS_currentStep:=SS_currentStep+1;			
				Led_Run:=FALSE;
				IF SS_currentStep=SS_StepNumber THEN								
					SS_MoveState:=88;
				END_IF
				IF SS_currentStep<SS_StepNumber THEN
					SS_MoveState:=77;
				END_IF
		77://等待单步时长够
				IF SS_TON.Q THEN
					SS_TON.IN:=FALSE;
					SS_MoveState:=0;
				END_IF
		88:
				SS_TON.IN:=FALSE;
				SS_Move:=FALSE;	
				Led_Run:=FALSE;
				SS_MoveState:=0;
				SS_currentStep:=0;
				SS_InitStartPositionDone:=FALSE;
				//SS_StepSystemTime[SS_StepNumber]:=F_GetSysTime();
	END_CASE
END_IF
(*获取每一步耗时*)
//FOR	m:= 0 TO SS_StepNumber DO
//	SS_StepCountTime[m]:=(SS_StepSystemTime_End[m]-SS_StepSystemTime_Begin[m]);
//END_FOR

(*STOP*)
IF SS_Stop OR btn_reset THEN
	FB_Move.BCGapReset:=TRUE;
	FB_Move();	
	SS_Move:=FALSE;	
	SS_MoveState:=0;	
	CASE SS_StopState OF
			0:
				FB_Stop.Mode:=5;						
				FB_Stop.CoupleState:=st_Couple;		
				FB_Stop.PowerState:=st_Power;			
				FB_Stop.BCGapStop:=TRUE;			
				FB_Stop();						
				SS_StopState:=1;
			1:
				FB_Stop();
				IF NOT FB_Stop.BCGapDone THEN		
					SS_StopState:=1;
				ELSE							
					SS_StopState:=88;
				END_IF
			88:
				SS_Stop:=FALSE;					
				FB_Move.BCGapReset:=FALSE;		
				SS_StopState:=0;
				btn_reset:=FALSE;
				//SS_Stop2:=FALSE;
		END_CASE
END_IF

(*触发限位开关后，相当于点击了Stop按钮*)
FTrig_ReachLS(CLK:=Unreach_LS_Far AND Unreach_LS_Near);
IF FTrig_ReachLS.Q THEN
	SS_Stop:=TRUE;
END_IF
END_ACTION

ACTION A_TaperMotionProtection:
(*如果该ID没有taper需求，则TaperFunctionSolidOn=FALSE，则判定taperOrNot和BLTaperOrNot都为FALSE*)
IF NOT TaperFunctionSolidOn THEN
	TaperOrNot:=FALSE;
	BLTaperOrNot:=FALSE;
END_IF
(*若GAP将有变化，首先检测TAPER是否超出阈值，若超出，则报错，提示必须先将TAPER回归到0，才可以改变GAP*)
IF NormalGapMode OR IDTaperMode THEN 
	IF NOT (Global_ChainProtection_MPS_Triggered OR Global_ChainProtection_EPS_Triggered) THEN//在触发联锁保护后，taper保护关闭
		IF ABS(UserGapPositionNew-UserGapPositionDisplay)>Threshold_GapChangeFlag AND btn_UserGapMove THEN
			IF UserTaperPositionDisplay>Threshold_TaperChangeFlag THEN
				btn_UserGapStop:=TRUE;
				btn_UserGapMove:=FALSE;
				Error:=TRUE;
				ErrorId:=809;
				ErrorDescription:='Please Move Taper to zero first before move gap';
				RETURN;
			END_IF
		END_IF
	END_IF
END_IF
IF BLTaperMode THEN
		IF NOT (Global_ChainProtection_MPS_Triggered OR Global_ChainProtection_EPS_Triggered) THEN//在触发联锁保护后，taper保护关闭
		IF ABS(UserGapPositionNew-UserGapPositionDisplay)>Threshold_GapChangeFlag AND btn_UserGapMove THEN
			IF BLUserTaperPositionDisplay>Threshold_TaperChangeFlag THEN
				btn_UserGapStop:=TRUE;
				btn_UserGapMove:=FALSE;
				Error:=TRUE;
				ErrorId:=810;
				ErrorDescription:='Please Move Taper to zero first before move gap';
				RETURN;
			END_IF
		END_IF
	END_IF
END_IF
(*若GAP将有变化,检测taper功能开关有没有关，要是没有关，提示先关闭*)
IF NOT (Global_ChainProtection_MPS_Triggered OR Global_ChainProtection_EPS_Triggered) THEN//在触发联锁保护后，taper保护关闭
	IF ABS(UserGapPositionNew-UserGapPositionDisplay)>Threshold_GapChangeFlag AND btn_UserGapMove THEN
		IF TaperOrNot OR BLTaperOrNot THEN
			btn_UserGapStop:=TRUE;
			btn_UserGapMove:=FALSE;
			Error:=TRUE;
			ErrorId:=811;
			ErrorDescription:='Please turn off taper function before move gap';
			RETURN;
		END_IF
	END_IF
END_IF
(*Taper和gap连锁限制性保护。比如11mm时候如果taper，入口端gap变小，会有压真空盒的问题。设置保护；在大间隙同样保护*)
IF IDTaperMode THEN
	IF NOT (Global_ChainProtection_MPS_Triggered OR Global_ChainProtection_EPS_Triggered)  THEN//在触发联锁保护后，taper保护关闭
		IF UserGapPositionNew-TaperAndGapSafetyfactor*TaperAndGapSafetyScale*UserTaperPositionNew<(min_UserGapPositionNew+TaperAndGapSafetyMinGapMargin)
			OR UserGapPositionNew+TaperAndGapSafetyfactor*TaperAndGapSafetyScale*UserTaperPositionNew>(max_UserGapPositionNew-TaperAndGapSafetyMinGapMargin) THEN
				 IF btn_UserGapMove THEN
					btn_UserGapStop:=TRUE;
					btn_UserGapMove:=FALSE;
					Error:=TRUE;
					ErrorId:=812;
					ErrorDescription:='Target taper is too big at current Gap';
					RETURN;
				END_IF
		END_IF
	END_IF
END_IF
IF BLTaperMode THEN
	IF NOT (Global_ChainProtection_MPS_Triggered OR Global_ChainProtection_EPS_Triggered)  THEN//在触发联锁保护后，taper保护关闭
		IF UserGapPositionNew-BLUserTaperPositionNew/2<(min_UserGapPositionNew+TaperAndGapSafetyMinGapMargin)
			OR UserGapPositionNew+BLUserTaperPositionNew/2>(max_UserGapPositionNew-TaperAndGapSafetyMinGapMargin) THEN
				 IF btn_UserGapMove THEN
					btn_UserGapStop:=TRUE;
					btn_UserGapMove:=FALSE;
					Error:=TRUE;
					ErrorId:=813;
					ErrorDescription:='Target taper is too big at current Gap';
					RETURN;
				END_IF
		END_IF
	END_IF
END_IF
(*Taper和gap连锁限制性保护。大间隙taper过大，有触碰真空盒问题，保护*)
END_ACTION

ACTION A_TaperParametersInit:
// 先做模式判断
NormalGapMode := NOT TaperOrNot AND NOT BLTaperOrNot;
IDTaperMode := TaperOrNot AND NOT BLTaperOrNot;
BLTaperMode := NOT TaperOrNot AND BLTaperOrNot;
//TaperOrNot和BLTaperOrNot互斥，只能选择其中一个
trig_TaperOrNot(CLK := TaperOrNot);
trig_BLTaperOrNot(CLK := BLTaperOrNot);
IF trig_TaperOrNot.Q THEN
    BLTaperOrNot := FALSE;
ELSIF trig_BLTaperOrNot.Q THEN
    TaperOrNot := FALSE;
END_IF;

//插入件taper/线站taper
IDTaperAndBLTaperScale:=L_Center2Motor/L_HalfGirder;
//插入件taper模式下，入口被动减小的距离，也即a
TaperAndGapSafetyScale:=(L_HalfGirder-L_Center2Motor)/(2*L_Center2Motor);

//线站模式下，最大taper由参数表决定，ID模式的最大tape由scale计算得到
max_UserTaperPositionNew:=max_BLUserTaperPositionNew*IDTaperAndBLTaperScale;
max_UserTaperVelocityNew:=max_BLUserTaperVelocityNew;
//最小taper固定位0
min_UserTaperPositionNew:=0;
min_UserTaperVelocityNew:=0;
END_ACTION

END_PROGRAM

(* stored: Version 1.1.0.1, ProductVersion 3.1.4024.6
   POU UserMode: Id {dbb58c86-3204-4c0e-a297-03b24a68bd10}, SpecialFunc None
   Action A_CheckCoupleStatus: Id {ec531655-4226-4156-a0f2-db7d67f06866}
   Action A_CheckMotorsPos: Id {f3cd81f2-82fa-493f-8c36-20c483307c7d}
   Action A_CryogenicChainProtection: Id {0f06233a-318c-40de-b717-6b9b4bac4cd3}
   Action A_GlobalChainProtection_EPS: Id {06b22d18-fd3c-40de-ae42-96c81b461f09}
   Action A_GlobalChainProtection_MPS: Id {214f7982-b3a1-46e2-bee6-e29b232f3cd2}
   Action A_InitCompensationData: Id {1e6a9c39-c8a5-4c48-b57c-71effe5e3747}
   Action A_MonitoringAllAxis: Id {ca11d2cd-2857-4b76-bcfc-746a563d8a76}
   Action A_OneKeyToMaxGap: Id {ba9dc3e9-1e8e-4d76-8af6-498bfc77c09c}
   Action A_OneKeyToTaperZero: Id {adaffbb5-af85-410b-b60e-03d094e0c42c}
   Action A_PowerOff: Id {e3ff8ae4-6e0c-4bb4-9a62-00e47841163f}
   Action A_PowerOn: Id {cacab3c1-f169-458e-acb8-60acf8e4d140}
   Action A_RegularMotion: Id {79d2706f-89ad-4612-adf2-c80c9fc85b18}
   Action A_SpectroscopyScanningMotion: Id {6676a965-5ff1-46e4-b651-02d2762b99bc}
   Action A_TaperMotionProtection: Id {70f980d5-eaf4-4284-9f18-474f849d8dc0}
   Action A_TaperParametersInit: Id {f7d8ca87-61a6-4e96-bac7-88c87690d17b} *)
